	IF TimeElapsed > 0 THEN
		Speed_ips := (Distance/TimeElapsed);
		Speed_fps := Speed_ips/12;
		Speed_fpm := Speed_fps*60;
	END_IF
	IF TotalCounts > 0 THEN
		DistperCount := Distance / UDINT_TO_REAL(TotalCounts);
	END_IF
		Reading := FALSE;
END_IF

END_PROGRAM

// ---- FunctionBlocks/Binder/BinderX_ReleaseControl.TcPOU
PROGRAM BinderX_ReleaseControl
VAR
	BinderHoldFB: FB_Binder_SingulateHold;
	Binder_Pusher: FB_BinderPusher;

	Binder		:	ST_Binder;

	BinderDataIn AT %I*: ST_FromBinder;
	BinderDataOut AT %Q*: ST_ToBinder;
	BinderState AT %I*: ST_BinderState;
	
	// Dummy Points for Compiling
	dummyIn		:	BOOL;
	dummyOut	:	BOOL;
	OCRHoldFB: INT;
END_VAR

VAR_OUTPUT
	Online	AT %Q*	: BOOL; // Send Online state to Safety
END_VAR

VAR CONSTANT
	GRABBER1_OCCUPIED:	UINT  := 1;
	GRABBER2_OCCUPIED: 	UINT  := 2;
	HOLDER_OCCUPIED:		UINT  := 3;
	PINSTOP_OUT:			UINT  := 4;
	
	PAUSED:						UINT  := 0;
	PRODUCT_PRESENT:			UINT  := 1;
	PRODUCT_ENTERING_OCR:		UINT  := 2;
	PRODUCT_READY_TO_PROCESS:	UINT  := 3;
	OCR_FINISHED:				UINT  := 4;	
	PRODUCT_EXITING_OCR:		UINT  := 5;
	RETURN_CONVEYOR_CLEARING:	UINT  := 6;
	RETURN_CONVEYOR_BUSY:		UINT  := 7;
END_VAR

(*
	Commented lines indicate what type of data item should be used for the signaling
*)

BinderHoldFB(
	In_Pause:= NOT Binder.FromBinder.Online,
//	In_ConveyorRunning := Conveyors.P8030_VFD.IsRunning,
	In_ReturnConveyorClearTime:= T#250MS, 
//	In_Grabber_Auto := Solenoids.GR8030_1_Status.Sts_EquipmentState.StsAuto,
//	In_GrabberExtended := ProxSensors.PX_23661_Extended.Out,
//	In_GrabberRetracted := ProxSensors.PX_23641_Retracted.Out,
//	In_SV_GrabberExtend := GVL_IO.SOL_10_Extend,
//	In_SV_GrabberRetract := GVL_IO.SOL_10_Retract,
//	In_PinStop_1_Auto := Solenoids.PS8030_1_Status.Sts_EquipmentState.StsAuto,
//	In_PinStop_1_Extended := ProxSensors.PX_23701_Extended.Out,
//	In_PinStop_1_Retracted := ProxSensors.PX_23681_Retracted.Out,
//	In_SV_PinStop_1_Extend := GVL_IO.SOL_11_Extend,
//	In_SV_PinStop_1_Retract := GVL_IO.SOL_11_Retract,
//	In_Holder_Auto := Solenoids.PS8030_2_Status.Sts_EquipmentState.StsAuto,
//	In_HolderExtended := ProxSensors.PX_23501_Extended.Out,
//	In_HolderRetracted := ProxSensors.PX_23481_Retracted.Out,
//	In_SV_HolderExtend := GVL_IO.SOL_13_Extend,
//	In_SV_HolderRetract := GVL_IO.SOL_13_Retract,
//	In_PinStop_2_Auto := Solenoids.PS8030_2_Status.Sts_EquipmentState.StsAuto,
//	In_PinStop_2_Extended := ProxSensors.PX_23541_Extended.Out,
//	In_PinStop_2_Retracted := ProxSensors.PX_23521_Retracted.Out,
//	In_SV_PinStop_2_Extend := GVL_IO.SOL_12_Extend,
//	In_SV_PinStop_2_Retract := GVL_IO.SOL_12_Retract,
	IN_Binder_Finished:= BinderDataIn.ProcessingComplete, 
//	PE_Grabber:= PhotoEyes.PE_23241.Out_OnOffFltrd, 
//	PE_PinStop_1:= PhotoEyes.PE_23461.Out_OnOffFltrd, 
//	PE_Holder:= PhotoEyes.PE_23521.Out_OnOffFltrd, 
//	PE_BinderExit := PhotoEyes.PE_23621.Out_OffFltrd, 
//	PE_ReturnConveyorOccupied:= PhotoEyes.PE_23741.Out_OffFltrd, 
	Status=> BinderDataOut.StatusSingulator, 
	Status_Output=> );

// Update variable to OCR that product is held and ready to be processed
//BinderDataOut.ProductHeld := BinderHoldFB.Status.PRODUCT_READY_TO_PROCESS AND GVL_IO.SOL_13_Extend AND ProxSensors.PX_23501_Extended.OutOnFltrd;;

// Push product out  
//Binder_Pusher(PE_Pusher:= (GVL_IO.P8030_Status.Sts_IsRunning) AND (PhotoEyes.PE_23621.Out) AND BinderHoldFB.Status.PRODUCT_EXITING_OCR,
//	PushTime:= T#250MS, 
//	);

//Binder.State.VlvBankPower := GVL_IO.OCRVlvBankPwr;
//Binder.State.DumpValve := GVL_IO.BinderAirDump; 
//Binder.State.SystemEstopOK := GVL_IO.SystemEstopsOK;
Binder.FromBinder := BinderDataIn;
Binder.ToBinder := BinderDataOut;

Online := BinderDataIn.Online;

END_PROGRAM

// ---- FunctionBlocks/Binder/FB_Binder_SingulateHold.TcPOU
FUNCTION_BLOCK FB_Binder_SingulateHold
VAR_INPUT
	{attribute 'OPC.UA.DA' := '1'}
	In_ResetState				:	BOOL;		// Clear the current functional state of the Binder

	In_Pause					:	BOOL;
	In_ConveyorRunning			:	BOOL;
	In_ReturnConveyorClearTime	:	TIME;
	IN_Binder_Finished			:	BOOL;
	
	PE_Grabber					:	BOOL;
	PE_PinStop_1				:	BOOL;
	PE_Holder					:	BOOL;
	PE_BinderExit				:	BOOL;
	PE_ReturnConveyorOccupied	:	BOOL;  // Photo eye that detects product on rack return conveyor
	
	In_Grabber_Auto				:	BOOL;
	In_SV_GrabberExtend			:	BOOL;
	In_SV_GrabberRetract		:	BOOL;
	In_GrabberExtended			:	BOOL;
	In_GrabberRetracted			:	BOOL;

	In_PinStop_1_Auto			:	BOOL;
	In_SV_PinStop_1_Extend		:	BOOL;
	In_SV_PinStop_1_Retract		:	BOOL;
	In_PinStop_1_Extended		:	BOOL;
	In_PinStop_1_Retracted		:	BOOL;

	In_PinStop_2_Auto			:	BOOL;
	In_SV_PinStop_2_Extend		:	BOOL;
	In_SV_PinStop_2_Retract		:	BOOL;
	In_PinStop_2_Extended		:	BOOL;
	In_PinStop_2_Retracted		:	BOOL;

	In_Holder_Auto				:	BOOL;
	In_SV_HolderExtend			:	BOOL;
	In_SV_HolderRetract			:	BOOL;
	In_HolderExtended			:	BOOL;
	In_HolderRetracted			:	BOOL;
	
END_VAR
VAR_OUTPUT
	{attribute 'OPC.UA.DA' := '1'}
	Out_Homed					:	BOOL;
	{attribute 'OPC.UA.DA' := '1'}
	Out_Ready					:	BOOL;
	{attribute 'OPC.UA.DA' := '1'}
	Out_Running					:	BOOL;

	Out_Grabber_Ext				:	BOOL;
	Out_Grabber_Ret				:	BOOL;

	Out_PinStop_1_Ext			:	BOOL;
	Out_PinStop_1_Ret			:	BOOL;

	Out_PinStop_2_Ext			:	BOOL;
	Out_PinStop_2_Ret			:	BOOL;

	Out_Holder_Ext				:	BOOL;
	Out_Holder_Ret				:	BOOL;
	
	{attribute 'OPC.UA.DA' := '1'}
	Status						:	UINT;		// General Binder singulate and hold status
	Status_Output				:	UINT;		// Binder singulate pin stop and grabber status
	
END_VAR
VAR	
	StartUp						:	BOOL := TRUE;
	rReturnConveyorOccupied		:	R_TRIG;
	fReturnConveyorExit			:	F_TRIG;
	tofReleaseConveyorClearTimer:	TOF;
	rProductFinished			:	R_TRIG;
	fProductCleared				:	F_TRIG;
	
	rProductEntering			:	R_TRIG;
	fProductEntering			:	F_TRIG;
	rResetState					:	R_TRIG;
	
	tonHomeWait					:	TON := (PT := T#1S);
	tonReadyWait				:	TON := (PT := T#1S);
	tonRunningWait				:	TON := (PT := T#5S);

	// Extend and Retract controls
	Grabber_Extend				:	BOOL;
	Grabber_Retract				:	BOOL;
	PinStop_1_Extend			:	BOOL;
	PinStop_1_Retract			:	BOOL;
	Holder_Extend				:	BOOL;
	Holder_Retract				:	BOOL;
	PinStop_2_Extend			:	BOOL;
	PinStop_2_Retract			:	BOOL;
END_VAR

VAR CONSTANT
	// Output Status
	GRABBER_OCCUPIED			:	UINT  := 1;
	PINSTOP_1_OUT				:	UINT  := 2;
	HOLDER_OCCUPIED				:	UINT  := 3;
	PINSTOP_2_OUT				:	UINT  := 4;
	
	// Singulation Status
	PAUSED						:	UINT  := 0;
	PRODUCT_PRESENT				:	UINT  := 1;
	PRODUCT_ENTERING_BINDER		:	UINT  := 2;
	PRODUCT_READY_TO_PROCESS	:	UINT  := 3;
	BINDER_FINISHED				:	UINT  := 4;	
	PRODUCT_EXITING_BINDER		:	UINT  := 5;
	RETURN_CONVEYOR_CLEARING	:	UINT  := 6;
	RETURN_CONVEYOR_BUSY		:	UINT  := 7;
END_VAR

// Process the In_ResetState
rResetState(CLK:=In_ResetState);

IF rResetState.Q THEN
	// Clear the Status
	Status := 0;
	// Revert to the StartUp state
	StartUp := TRUE;
	// Revert to the NOT Homed state
	Out_Homed := FALSE;
	tonHomeWait(IN := FALSE);
	// Revert to the NOT Ready state
	Out_Ready := FALSE;
	tonReadyWait(IN := FALSE);
	// Revert to the NOT Running state
	Out_Running := FALSE;
	tonRunningWait(IN := FALSE);
	// Clear the reset request
	In_ResetState := FALSE;
END_IF

// Home the 
IF StartUp  OR NOT Out_Homed OR NOT Out_Ready THEN
	Status.PAUSED := TRUE;
	
	tonHomeWait.IN := NOT Out_Homed;
	tonHomeWait();
	IF NOT Out_Homed THEN
		// Grabber
		Grabber_Retract := TRUE;
		Grabber_Extend := FALSE;
		// PinStop_1
		PinStop_1_Retract := FALSE;
		PinStop_1_Extend := TRUE;
		// Holder
		Holder_Retract := TRUE;
		Holder_Extend := FALSE;
		// PinStop_2
		PinStop_2_Retract := FALSE;
		PinStop_2_Extend := TRUE;
		IF In_GrabberRetracted
		   AND In_PinStop_1_Extended
		   AND In_HolderRetracted
		   AND In_PinStop_2_Extended
		   THEN
			Out_Homed := tonHomeWait.Q;
		END_IF
	END_IF

	tonReadyWait.IN := NOT Out_Ready AND Out_Homed;
	tonReadyWait();
	IF NOT Out_Ready AND Out_Homed THEN
		// PinStop_1
		PinStop_1_Retract := FALSE;
		PinStop_1_Extend := TRUE;
		// PinStop_2
		PinStop_2_Retract := FALSE;
		PinStop_2_Extend := TRUE;
		IF In_GrabberRetracted
		   AND In_PinStop_1_Extended
		   AND In_HolderRetracted
		   AND In_PinStop_2_Extended
		   THEN
			Out_Ready := tonReadyWait.Q;
		END_IF
	END_IF

	StartUp := NOT Out_Homed OR NOT Out_Ready;
	Out_Running := FALSE;
	
ELSIF In_Pause OR NOT In_ConveyorRunning THEN
	// Grabber
	Grabber_Retract := FALSE;
	Grabber_Extend := FALSE;
	// PinStop_1
	PinStop_1_Retract := FALSE;
	PinStop_1_Extend := FALSE;
	// Holder
	Holder_Retract := FALSE;
	Holder_Extend := FALSE;
	// PinStop_2
	PinStop_2_Retract := FALSE;
	PinStop_2_Extend := FALSE;

ELSIF NOT Out_Running THEN
	tonRunningWait.IN := NOT OUT_Running AND Out_Ready AND Out_Homed AND In_ConveyorRunning;
	tonRunningWait();
	Out_Running := tonRunningWait.Q;
ELSIF Out_Running THEN
	Status.PAUSED := FALSE;

	a_EntryControl();
		
	a_ReleaseToBinder();
	
	a_HoldProduct();
	
	// Watch finished trigger to release product from
	rProductFinished(CLK:= IN_Binder_Finished);
	
	IF rProductFinished.Q THEN
		Status.BINDER_FINISHED := TRUE;
	END_IF
	
	// Watch release conveyor to make sure it is clear to release from OCR
	a_WatchReleaseConveyor();
		
	a_ReleaseFromBinder();
	
	fProductCleared(CLK:= PE_BinderExit AND Status.PRODUCT_EXITING_BINDER);
	
	// PinStop_2
	PinStop_2_Retract := Status.PRODUCT_EXITING_BINDER;
	PinStop_2_Extend := NOT Status.PRODUCT_EXITING_BINDER;
	IF fProductCleared.Q THEN
		Status.PRODUCT_EXITING_BINDER := FALSE;
//		IF Status.PRODUCT_PRESENT OR PE_PinStop_1 THEN
//			ReleaseToOCR();
//		END_IF
	END_IF
ELSE
	// Grabber
	Grabber_Retract := TRUE;
	Grabber_Extend := FALSE;
	// PinStop_1
	PinStop_1_Retract := FALSE;
	PinStop_1_Extend := TRUE;
	// Holder
	Holder_Retract := TRUE;
	Holder_Extend := FALSE;
	// PinStop_2
	PinStop_2_Retract := FALSE;
	PinStop_2_Extend := TRUE;
END_IF

// Activate all the outputs in one place
Status_Output.GRABBER_OCCUPIED := Grabber(Active := In_Grabber_Auto, Extend:= Grabber_Extend, Retract := Grabber_Retract);
Status_Output.HOLDER_OCCUPIED := Holder(Active := In_Holder_Auto, Extend:= Holder_Extend, Retract := Holder_Retract);
Status_Output.PINSTOP_1_OUT := PinStop_1(Active:= In_PinStop_1_Auto, Extend := PinStop_1_Extend, Retract:= PinStop_1_Retract);
Status_Output.PINSTOP_2_OUT := PinStop_2(Active:= In_PinStop_2_Auto, Extend := PinStop_2_Extend, Retract:= PinStop_2_Retract);

ACTION a_EntryControl:
(* Set PRODUCT_PRESENT when:
	PE_PinStop_1 is ON
	OR PRODUCT_ENTERRING_OCR is ON
*)
Status.PRODUCT_PRESENT := PE_PinStop_1 OR Status.PRODUCT_ENTERING_BINDER;
// Retract the Pin stop in response to the Release to the OCR, and the state of the Pin stop PE
rProductEntering(CLK:= Status.PRODUCT_ENTERING_BINDER);
IF rProductEntering.Q THEN
	PinStop_1_Extend := FALSE;
	PinStop_1_Retract := TRUE;
END_IF
fProductEntering(CLK := PE_PinStop_1);
IF fProductEntering.Q THEN
	PinStop_1_Extend := TRUE;
	PinStop_1_Retract := FALSE;
END_IF

// If the grabber recieves product while Product is physically or logically at Pin Stop 1, then hold it at the grabber

Grabber_Extend := (PE_Grabber AND Status.PRODUCT_PRESENT) OR Status.PRODUCT_ENTERING_BINDER;
Grabber_Retract := NOT Grabber_Extend;
END_ACTION

ACTION a_HoldProduct:
IF PE_Holder THEN
	Status.PRODUCT_PRESENT := FALSE;
	Status.PRODUCT_ENTERING_BINDER := FALSE;
	IF NOT Status.PRODUCT_EXITING_BINDER THEN
		Holder_Extend := TRUE;
		Holder_Retract := FALSE;
		Status.PRODUCT_READY_TO_PROCESS := TRUE;
	END_IF
END_IF
END_ACTION

ACTION a_ReleaseFromBinder:
IF Status.BINDER_FINISHED AND NOT(Status.RETURN_CONVEYOR_BUSY) THEN
	Status.PRODUCT_READY_TO_PROCESS := FALSE;
	Status.PRODUCT_EXITING_BINDER := TRUE;
	Status.BINDER_FINISHED := FALSE;
	// Holder
	Holder_Retract := TRUE;
	Holder_Extend := FALSE;
	// PinStop_2
	PinStop_2_Retract := TRUE;
	PinStop_2_Extend := FALSE;
END_IF
END_ACTION

ACTION a_ReleaseToBinder:
IF Status.PRODUCT_PRESENT 
   AND NOT(Status_Output.HOLDER_OCCUPIED)
   AND NOT(Status.PRODUCT_ENTERING_BINDER)
   AND NOT(Status.PRODUCT_EXITING_BINDER)  THEN
	Status.PRODUCT_ENTERING_BINDER := TRUE;
END_IF
END_ACTION

ACTION a_WatchReleaseConveyor:
rReturnConveyorOccupied(CLK:= PE_ReturnConveyorOccupied);

IF rReturnConveyorOccupied.Q THEN
	Status.RETURN_CONVEYOR_CLEARING := TRUE;
END_IF

fReturnConveyorExit(CLK:= Status.RETURN_CONVEYOR_BUSY AND PE_BinderExit);

IF fReturnConveyorExit.Q THEN
	Status.RETURN_CONVEYOR_CLEARING := FALSE;
END_IF

tofReleaseConveyorClearTimer(IN:= Status.RETURN_CONVEYOR_CLEARING, PT:= In_ReturnConveyorClearTime);

Status.RETURN_CONVEYOR_BUSY:= tofReleaseConveyorClearTimer.Q;
END_ACTION

METHOD Grabber : BOOL
VAR_INPUT
	Active	: BOOL;	
	Extend	: BOOL;
	Retract	: BOOL;
END_VAR
IF Active THEN
	IF Extend THEN
		Out_Grabber_Ext := TRUE;
		Out_Grabber_Ret := FALSE;
	ELSIF Retract THEN
		Out_Grabber_Ext := FALSE;
		Out_Grabber_Ret := TRUE;
	ELSE
		Out_Grabber_Ext := FALSE;
		Out_Grabber_Ret := FALSE;
	END_IF
ELSE
	Out_Grabber_Ext := FALSE;
	Out_Grabber_Ret := FALSE;
END_IF

Grabber := Out_Grabber_Ext OR In_GrabberExtended;
END_METHOD

METHOD Holder : BOOL
VAR_INPUT
	Active	: BOOL;
	Extend	: BOOL;
	Retract	: BOOL;
END_VAR
IF Active THEN
	IF Extend THEN
		Out_Holder_Ext := TRUE;
		Out_Holder_Ret := FALSE;
	ELSIF Retract THEN
		Out_Holder_Ext := FALSE;
		Out_Holder_Ret := TRUE;
	ELSE
		Out_Holder_Ext := FALSE;
		Out_Holder_Ret := FALSE;
	END_IF
ELSE
	Out_Holder_Ext := FALSE;
	Out_Holder_Ret := FALSE;
END_IF

Holder := Out_Holder_Ext OR In_HolderExtended;
END_METHOD

METHOD PinStop_1 : BOOL
VAR_INPUT
	Active	: BOOL;	
	Extend	: BOOL;
	Retract	: BOOL;
END_VAR
IF Active THEN
	IF Extend THEN
		Out_PinStop_1_Ext := TRUE;
		Out_PinStop_1_Ret := FALSE;
	ELSIF Retract THEN
		Out_PinStop_1_Ext := FALSE;
		Out_PinStop_1_Ret := TRUE;
	ELSE
		Out_PinStop_1_Ext := FALSE;
		Out_PinStop_1_Ret := FALSE;
	END_IF
ELSE
	Out_PinStop_1_Ext := FALSE;
	Out_PinStop_1_Ret := FALSE;
END_IF

PinStop_1 := Out_PinStop_1_Ext OR In_PinStop_1_Extended;
END_METHOD

METHOD PinStop_2 : BOOL
VAR_INPUT
	Active	: BOOL;
	Extend	: BOOL;
	Retract	: BOOL;
END_VAR
IF Active THEN
	IF Extend THEN
		Out_PinStop_2_Ext := TRUE;
		Out_PinStop_2_Ret := FALSE;
	ELSIF Retract THEN
		Out_PinStop_2_Ext := FALSE;
		Out_PinStop_2_Ret := TRUE;
	ELSE
		Out_PinStop_2_Ext := FALSE;
		Out_PinStop_2_Ret := FALSE;
	END_IF
ELSE
	Out_PinStop_2_Ext := FALSE;
	Out_PinStop_2_Ret := FALSE;
END_IF

PinStop_2 := Out_PinStop_2_Ext OR In_PinStop_2_Extended;
END_METHOD

END_FUNCTION_BLOCK

// ---- FunctionBlocks/Binder/FB_BinderPusher.TcPOU
FUNCTION_BLOCK FB_BinderPusher
VAR_INPUT
	PE_Pusher: BOOL;
	PushTime:	TIME;
END_VAR
VAR_OUTPUT
	Out_Pusher_Ext:	BOOL;
	Out_Pusher_Ret:	BOOL;
	PushingActive: BOOL;
END_VAR
VAR
	fPusher: F_TRIG;
	
	tonPusherArm: TON;
END_VAR

fPusher(CLK:= PE_Pusher);

IF fPusher.Q THEN
	Out_Pusher_Ext := TRUE;
	Out_Pusher_Ret := FALSE;
	PushingActive := TRUE;
END_IF

tonPusherArm(IN:=PushingActive , PT:= PushTime);

IF tonPusherArm.Q  THEN
	Out_Pusher_Ext := FALSE;
	Out_Pusher_Ret := TRUE;
	PushingActive := FALSE;
END_IF

END_FUNCTION_BLOCK

// ---- FunctionBlocks/FB_Merge/FB_Merge2.TcPOU
FUNCTION_BLOCK FB_Merge2
(* This function block can handle any number of Inlets to the merge by changing the constant "Cfg_MergeInletCount" 
	and then saving it as a new named function block. 
*)

VAR CONSTANT
	MERGEINLETCOUNT			:	INT := 2;		// Number of inlets on the merge
END_VAR

VAR_IN_OUT
	In_MergeProcessOrder	:	ARRAY [1..MERGEINLETCOUNT] OF INT;	// Processing order of the merge inlets
END_VAR

VAR_INPUT
	{attribute 'OPC.UA.DA' := '1'}
	In_MergeState				:	E_StateCntrl;	// The State of the merge take away conveyor
	In_MergeInletArry			:	ARRAY [1..MERGEINLETCOUNT] OF ST_MergeInlet;
	In_MergeTakeAwayMtrFdbk		:	BOOL;			// Merge Take Away Motor Feedback, 1=Running
	{attribute 'OPC.UA.DA' := '1'}
	In_PhotoEyeJamDetect		:	BOOL;			// Photo Eye located to detect jams at the assigned merge
	
	In_SimActive				:	BOOL;	
	In_Init						:	BOOL;
		
	In_MergeWakeTrigArry		: 	ARRAY [1..5] OF BOOL;
	Cfg_ClearTakeAwayTime		: 	REAL;
	{attribute 'OPC.UA.DA' := '1'}
	Cfg_MergeName				:	STRING(20);		// Name used to Identify the Merge on the HMI
	{attribute 'OPC.UA.DA' := '1'}
	Cfg_JammedTime				: 	REAL := 15;
END_VAR

VAR_OUTPUT
	Sts_MergeSts			:	ST_MergeSts;
	Sts_MergeInletStsArry	:	ARRAY [1..MERGEINLETCOUNT]OF ST_MergeInletSts;
END_VAR

VAR
	MergeRunOutActive		:	BOOL;
	MergeStateChanged		:	R_TRIG;	
	LastMergeState			: 	E_StateCntrl;

	MergeEnabledRTrig		: 	R_TRIG;
	MergeEnabledFTrig		: 	F_TRIG;
	inletindex				: 	INT := 0;
	processIndex			:	INT := 0;	
	i						:	INT;
	j						:	INT;
	fb_MergeEntryArry		:	ARRAY [1..MERGEINLETCOUNT]OF FB_MergeInlet;
	MergeGrantedOwner		:	INT := 0;	// The ID (index) of the inlet that has the merge granted control 
	MergeSubState_old		: 	INT;
	AnotherMergeReqIsWaiting: 	BOOL;
	HiHiMergeReqIsWaiting	: 	BOOL;
	HiHiIndex				: 	INT;
	MergeCntrl				: 	INT;

	ClearTakeawayDelay		: 	BOOL;
	ClearTakeAwayTimer		: 	TON;
	LastClearTakeAwayTime	: 	REAL;
	nClearTakeAwayTime		: 	UINT;
	tClearTakeAwayTime		: 	TIME;

	LastJammedTime			:	REAL;
	nJammedTime				:	UINT;
	tJammedTime				:	TIME;
	fb_JamDetect			:	FB_JamDetect;
	
	bIncIndex				:	BOOL;
END_VAR

// Initialize the Merge Here
IF In_Init THEN
	// Make sure the Processing Order doesn't have zeros in it
	FOR i := 1 TO MERGEINLETCOUNT DO
		IF In_MergeProcessOrder[i] = 0 THEN
			In_MergeProcessOrder[i] := i;
		END_IF
	END_FOR
	IF processIndex = 0 THEN
		processIndex := 1;
	END_IF
	Sts_MergeSts.MergeSubState := E_MergeState.stStopped;
	Sts_MergeSts.MergeSubStateTxt := 'Stopped';
	Sts_MergeSts.InletCount := MERGEINLETCOUNT;
	MergeGrantedOwner := In_MergeProcessOrder[1];
END_IF

// Calculate and set the timer values
// Clear take away timer
IF LastClearTakeAwayTime <> Cfg_ClearTakeAwayTime THEN
	LastClearTakeAwayTime := Cfg_ClearTakeAwayTime;
	nClearTakeAwayTime := REAL_TO_UINT(LastClearTakeAwayTime * 1000); 
	tClearTakeAwayTime := UINT_TO_TIME(nClearTakeAwayTime);
END_IF

// Product Jam Wait timer
IF LastJammedTime <> Cfg_JammedTime THEN
	LastJammedTime := Cfg_JammedTime;
	nJammedTime := REAL_TO_UINT(LastJammedTime * 1000); 
	tJammedTime := UINT_TO_TIME(nJammedTime);
END_IF

// Run the Jam Detection
fb_JamDetect(In_PE := In_PhotoEyeJamDetect
			, In_Status := Sts_MergeSts.MergeTakeAwayMtrActive
			, CFG_PEOKState := 0
			, JamDetTime := tJammedTime
			, JamDetected => Sts_MergeSts.MergeJammed);

// Set MergeEnabled to the Take Away conveyor Auto, or the take away running, for manual opertion
Sts_MergeSts.MergeEnabled := ((In_MergeState = E_StateCntrl.stAuto) OR In_MergeTakeAwayMtrFdbk);

// If merge is just enabled set operation
MergeEnabledRTrig(CLK:= Sts_MergeSts.MergeEnabled, Q=> );	

// Cause a Re-process of the state when the state changes
MergeStateChanged(CLK := (In_MergeState <> LastMergeState), Q=> );
// Capture the state change for the next pass 
LastMergeState := In_MergeState;

// Test for a Merge state change, or an enable trigger
IF MergeEnabledRTrig.Q OR MergeStateChanged.Q THEN
	CASE In_MergeState OF
		// Auto
		E_StateCntrl.stAuto:
			Sts_MergeSts.MergeSubState := E_MergeState.stClearTakeAway;
			Sts_MergeSts.MergeSubStateTxt := 'Clear Take Away';
		
		// Manual
		E_StateCntrl.stManual:
			Sts_MergeSts.MergeTakeAwayMtrActive := In_MergeTakeAwayMtrFdbk;
			inletindex := DINT_TO_INT(In_MergeProcessOrder[1]);
			Sts_MergeSts.MergeSubState := E_MergeState.stMergeManual;
			Sts_MergeSts.MergeSubStateTxt := 'Manual';
	END_CASE
END_IF

// If Merge enabled drops set states per condition
MergeEnabledFTrig(CLK:= Sts_MergeSts.MergeEnabled, Q=> );
IF  MergeEnabledFTrig.Q OR MergeStateChanged.Q THEN
	CASE In_MergeState OF
		// Offline
		E_StateCntrl.stOffline:
			Sts_MergeSts.MergeSubState := E_MergeState.stStopped;
			Sts_MergeSts.MergeSubStateTxt := 'Stopped';
		// Faulted
		E_StateCntrl.stFaulted:
			Sts_MergeSts.MergeSubState := E_MergeState.stStopped;
			Sts_MergeSts.MergeSubStateTxt := 'Faulted';
	END_CASE
END_IF

//  ===== Set Up Merge Control for merge sub parts =====

// Call inlet function blocks
FOR i := 1 TO MERGEINLETCOUNT DO
	fb_MergeEntryArry[i](In_MergeSubState:= Sts_MergeSts.MergeSubState, In_TakeAwayMtrSts:= Sts_MergeSts.MergeTakeAwayMtrActive, In_MergeInletInput:= In_MergeInletArry[i], Sts_MergeInlet=> Sts_MergeInletStsArry[i], In_MergeWakeTrig := In_MergeWakeTrigArry[i]);
END_FOR

// Turn OFF the increment Index boolean
bIncIndex := FALSE;

CASE Sts_MergeSts.MergeSubState OF	
	// Stopped
	E_MergeState.stStopped:
		Sts_MergeSts.MergeTakeAwayMtrActive := FALSE;
		
	// Clear Takeaway	
	E_MergeState.stClearTakeAway:
		ClearTakeawayDelay := TRUE;
		// Set Take Away Motor Output
		Sts_MergeSts.MergeTakeAwayMtrActive := ClearTakeawayDelay;
		
	
		IF ClearTakeAwayTimer.Q THEN
			ClearTakeawayDelay := FALSE;
			//MergeGrantedOwner := 0;
			MergeGrantedOwner := In_MergeProcessOrder[1];
			// Reset Inlets and merge
			FOR i := 1 TO MERGEINLETCOUNT DO
				fb_MergeEntryArry[i].In_MergeGranted := FALSE;
			END_FOR
			 fb_MergeEntryArry[1].In_MergeGranted := TRUE;
			IF processIndex = 0 THEN
				processIndex := 1;
			END_IF
			inletindex := In_MergeProcessOrder[processIndex];
			Sts_MergeSts.MergeSubState := E_MergeState.stMergeOperational;
			Sts_MergeSts.MergeSubStateTxt := 'Operational';
		END_IF
		
	// Operational
	E_MergeState.stMergeOperational:

		// Set the inletIndex to the inlet identified at the processIndex in the ProcessOrder
		inletindex := In_MergeProcessOrder[processIndex];

		// Set Take Away Motor Output
		Sts_MergeSts.MergeTakeAwayMtrActive := TRUE;
		
		// Clear the flags that may be set
		AnotherMergeReqIsWaiting := FALSE;
		HiHiMergeReqIsWaiting := FALSE;
		HiHiIndex := 0;
		MergeRunOutActive := FALSE;
		FOR j := 1 TO MERGEINLETCOUNT DO
			IF fb_MergeEntryArry[j].Sts_MergeInlet.MergeRequested AND MergeGrantedOwner <> j AND MergeGrantedOwner <> 0 THEN
				AnotherMergeReqIsWaiting := TRUE;
			END_IF
			IF fb_MergeEntryArry[j].Sts_MergeInlet.HiHiDetected THEN
				HiHiMergeReqIsWaiting := TRUE;
				HiHiIndex := j;
			END_IF
			IF fb_MergeEntryArry[j].Sts_MergeInlet.MergeRunOutActive THEN
				MergeRunOutActive := TRUE;
			END_IF
		END_FOR

		// Call individual merge inlets branches
		IF fb_MergeEntryArry[inletindex].Sts_MergeInlet.MergeRequested THEN
			// Prioritize the HiHi request
			IF HiHiMergeReqIsWaiting THEN
				IF inletindex <> HiHiIndex THEN
					inletindex := HiHiIndex;
				END_IF
			END_IF
			IF NOT MergeRunOutActive THEN
				IF (MergeGrantedOwner = 0) THEN
					MergeGrantedOwner := inletindex;
					fb_MergeEntryArry[inletindex].In_MergeGranted := TRUE;
				END_IF
			END_IF
		ELSE
			bIncIndex := TRUE;
		END_IF	
		IF MergeGrantedOwner <> 0 THEN	
			IF (AnotherMergeReqIsWaiting AND fb_MergeEntryArry[MergeGrantedOwner].Sts_MergeInlet.MergeComplete)
			   OR HiHiMergeReqIsWaiting
			   THEN
				// Reset Inlet and merge
				fb_MergeEntryArry[MergeGrantedOwner].In_MergeGranted := FALSE;
				MergeGrantedOwner := 0;
				bIncIndex := TRUE;
			END_IF
		END_IF
	// Manual mode	
	E_MergeState.stMergeManual:
		// Set the inletIndex to the inlet identified at the processIndex in the ProcessOrder
		inletindex := In_MergeProcessOrder[processIndex];

		// Set Take Away Motor Output
		Sts_MergeSts.MergeTakeAwayMtrActive := In_MergeTakeAwayMtrFdbk;
		
		// Call individual merge inlets branches
		IF fb_MergeEntryArry[inletindex].Sts_MergeInlet.MergeRequested THEN
			// Prioritize the HiHi request
			IF HiHiMergeReqIsWaiting THEN
				IF inletindex <> HiHiIndex THEN
					inletindex := HiHiIndex;
				END_IF
			END_IF
			IF NOT MergeRunOutActive THEN
				IF (MergeGrantedOwner = 0) THEN
					MergeGrantedOwner := inletindex;
					fb_MergeEntryArry[inletindex].In_MergeGranted := TRUE;
				END_IF
			END_IF
		ELSE
			bIncIndex := TRUE;
		END_IF		
		IF (AnotherMergeReqIsWaiting AND fb_MergeEntryArry[MergeGrantedOwner].Sts_MergeInlet.MergeComplete)
			   OR HiHiMergeReqIsWaiting
			   THEN
				// Reset Inlet and merge
				fb_MergeEntryArry[MergeGrantedOwner].In_MergeGranted := FALSE;
				MergeGrantedOwner := 0;
				bIncIndex := TRUE;
		END_IF
END_CASE

// Take Away Timer
ClearTakeAwayTimer(IN:= ClearTakeawayDelay, PT:= tClearTakeAwayTime, Q=> , ET=> );

// Increment the processIndex
IF bIncIndex THEN
	processIndex := processIndex + 1;
	bIncIndex := FALSE;
	// Reset index if necessary
	IF (processIndex > MERGEINLETCOUNT) THEN
		processIndex := 1;
	END_IF
END_IF

END_FUNCTION_BLOCK

// ---- FunctionBlocks/FB_Merge/Merge Inlet/FB_MergeInlet.TcPOU
FUNCTION_BLOCK FB_MergeInlet
VAR_INPUT
	In_MergeSubState		:	E_MergeState;
	In_TakeAwayMtrSts		:	BOOL;
	In_MergeInletInput		:	ST_MergeInlet;	
	In_MergeGranted			:	BOOL;		// Merge request has been accepted and allowed (1=merge allowed)
	In_MergeWakeTrig		:   BOOL;
END_VAR
VAR_OUTPUT
	Sts_MergeInlet			:	ST_MergeInletSts;
END_VAR
VAR
	MergeEntryHasProduct		: 	BOOL;
	MergeEntryHighTimer			: 	TON;		// Timer to watch High Photo Eye
	MergeEntryHiHiTimer			: 	TON;		// Timer to watch HiHi Photo Eye
	MergeRelPrdctWaitTimer		: 	TON;		// Timer to release product if waiting too long for full mark to be reached
	
	InletStateChanged			:	R_TRIG;	
	LastInletState				: 	E_StateCntrl;
	InletEnabled				:	BOOL;

	ProductReleaseCountFTrig	: 	F_Trig;
	ReleaseCountWaitTimer		: 	TON;
	ClearRunOutTimer			: 	TP;			// Run the timer for this long to clear out the merge
	fClearRunOut				:	F_TRIG;		// Detect when the ClearRunOut has completed
	ClearHiHiTimer				: 	TP;			// Run the timer for this long to clear a HiHi condition
	MergeRequestRTrig			: 	R_TRIG;
	RunEnable					: 	BOOL;
	MergePreLoad				: 	BOOL;
	MergeGrantedFTrig			: 	F_TRIG;
	ManualModeFTrig				: 	F_TRIG;
	ManualOperEnable			: 	BOOL;
	ManModeTrig					: 	R_TRIG;
	TimerReleaseCountWaitActive	:	BOOL;
	LastHighTriggerTime			:	REAL;
	LastHiHiTriggerTime			:	REAL;
	LastHiHiClearTime			:	REAL;
	LastMrgReqPrdctWaitTime		:	REAL;
	LastReleaseCountWaitTime	:	REAL;
	LastClearRunOutTime			:	REAL;

	nHighTriggerTime			:	UINT;
	nHiHiTriggerTime			:	UINT;
	nHiHiClearTime				:	UINT;
	nMrgReqPrdctWaitTime		:	UINT;
	nReleaseCountWaitTime		:	UINT;
	nClearRunOutTime			:	UINT;

	tHighTriggerTime			:	TIME;
	tHiHiTriggerTime			:	TIME;
	tHiHiClearTime				:	TIME;
	tMrgReqPrdctWaitTime		:	TIME;
	tReleaseCountWaitTime		:	TIME;
	tClearRunOutTime			:	TIME;
END_VAR

// Calculate and set the timer values
// High Water Mark trigger timer
IF LastHighTriggerTime <> In_MergeInletInput.Cfg.Cfg_HighTriggerTime THEN
	LastHighTriggerTime := In_MergeInletInput.Cfg.Cfg_HighTriggerTime;
	nHighTriggerTime := REAL_TO_UINT(LastHighTriggerTime * 1000); 
	tHighTriggerTime := UINT_TO_TIME(nHighTriggerTime);
END_IF

// HiHi Water Mark trigger timer
IF LastHiHiTriggerTime <> In_MergeInletInput.Cfg.Cfg_HiHiTriggerTime THEN
	LastHiHiTriggerTime := In_MergeInletInput.Cfg.Cfg_HiHiTriggerTime;
	nHiHiTriggerTime := REAL_TO_UINT(LastHiHiTriggerTime * 1000); 
	tHiHiTriggerTime := UINT_TO_TIME(nHiHiTriggerTime);
END_IF

// HiHi Water Mark clear timer
IF LastHiHiClearTime <> In_MergeInletInput.Cfg.Cfg_HiHiClearTime THEN
	LastHiHiClearTime := In_MergeInletInput.Cfg.Cfg_HiHiClearTime;
	nHiHiClearTime := REAL_TO_UINT(LastHiHiClearTime * 1000); 
	tHiHiClearTime := UINT_TO_TIME(nHiHiClearTime);
END_IF

// Product Wait timer
IF LastMrgReqPrdctWaitTime <> In_MergeInletInput.Cfg.Cfg_MrgReqPrdctWaitTime THEN
	LastMrgReqPrdctWaitTime := In_MergeInletInput.Cfg.Cfg_MrgReqPrdctWaitTime;
	nMrgReqPrdctWaitTime := REAL_TO_UINT(LastMrgReqPrdctWaitTime * 1000); 
	tMrgReqPrdctWaitTime := UINT_TO_TIME(nMrgReqPrdctWaitTime);
END_IF

// Fulfilled Release Count Wait timer
IF LastReleaseCountWaitTime <> In_MergeInletInput.Cfg.Cfg_ReleaseCountWaitTime THEN
	LastReleaseCountWaitTime := In_MergeInletInput.Cfg.Cfg_ReleaseCountWaitTime;
	nReleaseCountWaitTime := REAL_TO_UINT(LastReleaseCountWaitTime * 1000); 
	tReleaseCountWaitTime := UINT_TO_TIME(nReleaseCountWaitTime);
END_IF

// Run-Out Clear timer
IF LastClearRunOutTime <> In_MergeInletInput.Cfg.Cfg_ClearRunOutTime THEN
	LastClearRunOutTime := In_MergeInletInput.Cfg.Cfg_ClearRunOutTime;
	nClearRunOutTime := REAL_TO_UINT(LastClearRunOutTime * 1000); 
	tClearRunOutTime := UINT_TO_TIME(nClearRunOutTime);
END_IF

// Set InletEnabled to the Inlet conveyor Auto, or the Inlet conveyor running (for manual opertion)
InletEnabled := ((In_MergeInletInput.Ctrl.In_InletState = E_StateCntrl.stAuto)
				OR (In_MergeInletInput.Ctrl.In_InletState = E_StateCntrl.stManual AND In_MergeInletInput.Ctrl.In_oMergeRelease));

// Watch for manual mode and manual PB
IF In_MergeSubState = E_MergeState.stMergeManual AND InletEnabled THEN
	ManualOperEnable := In_MergeInletInput.Ctrl.In_oMergeRelease;
ELSE
	ManualOperEnable := FALSE;
END_IF

ManualModeFTrig(CLK:= ManualOperEnable, Q=> );

// Look at photo eyes and determine if a merge request is needed
MergeEntryHasProduct:= (In_MergeSubState = E_MergeState.stMergeOperational)
 						AND In_MergeInletInput.Ctrl.PhotoEyeDischarge
						AND (In_MergeInletInput.Ctrl.In_InletState = E_StateCntrl.stAuto);
// Set timer to keep product from waiting too long if full mark is not met
MergeRelPrdctWaitTimer(IN:= MergeEntryHasProduct AND (In_MergeInletInput.Cfg.Cfg_UseHighWaterPE OR In_MergeInletInput.Cfg.Cfg_UseHiHiWaterPE)
						, PT:= tMrgReqPrdctWaitTime, Q=> , ET=> );

// Watch the Timer to check for a High Water event
MergeEntryHighTimer.IN:= In_MergeInletInput.Ctrl.PhotoEyeEntryHigh AND In_MergeInletInput.Cfg.Cfg_UseHighWaterPE AND MergeEntryHasProduct;
MergeEntryHighTimer(PT:= tHighTriggerTime, Q=> , ET=> );

// Watch the Timer to check for a HiHi Water event
MergeEntryHighTimer.IN:= In_MergeInletInput.Ctrl.PhotoEyeEntryHiHi AND In_MergeInletInput.Cfg.Cfg_UseHiHiWaterPE AND MergeEntryHasProduct;
MergeEntryHiHiTimer(PT:= tHiHiTriggerTime, Q=> , ET=> );
IF (MergeEntryHiHiTimer.Q) THEN
	Sts_MergeInlet.HiHiDetected := MergeEntryHiHiTimer.Q;
END_IF

// Set merge request based on entry and full PE's and wait timer(s)
IF ((MergeEntryHighTimer.Q)
   OR (MergeEntryHiHiTimer.Q)
   OR ((NOT In_MergeInletInput.Cfg.Cfg_UseHighWaterPE AND NOT In_MergeInletInput.Cfg.Cfg_UseHiHiWaterPE) AND MergeEntryHasProduct)
   OR (MergeRelPrdctWaitTimer.Q)) 
   AND (NOT Sts_MergeInlet.MergeRequested AND NOT In_MergeGranted) OR ManualOperEnable THEN
	Sts_MergeInlet.MergeRequested := TRUE;
ELSIF Sts_MergeInlet.MergeRequested AND (NOT MergeEntryHasProduct) AND (NOT In_MergeGranted) THEN
	Sts_MergeInlet.MergeRequested := FALSE;
ELSIF In_MergeGranted THEN
	Sts_MergeInlet.MergeRequested := FALSE;
END_IF

// Upon merge request or entry of manual mode reset Count, Timer and Complete bit
ManModeTrig(CLK:= In_MergeSubState = E_MergeState.stMergeManual, Q=> );
MergeRequestRTrig(CLK:= Sts_MergeInlet.MergeRequested, Q=> );
IF MergeRequestRTrig.Q OR ManModeTrig.Q THEN
	Sts_MergeInlet.CrrntReleaseCount := 0;
	Sts_MergeInlet.MergeComplete := FALSE;
//	ManualOperEnable := FALSE;
END_IF

// If merge granted and HiHi Water mark detected, run the merge for the HiHi Clear time
//	This is a Timer Pulse so it will run for a specified period of time after the rising edge of the In condition is detected 
ClearHiHiTimer(IN := Sts_MergeInlet.HiHiDetected AND In_MergeGranted, PT := tHiHiClearTime);
	
// If merge granted count product release on falling trigger of the photo eye
//	Don't add up the count if the ClearRunOutTimer is running
ProductReleaseCountFTrig(CLK:= In_MergeInletInput.Ctrl.PhotoEyeDischarge, Q=> );
IF ProductReleaseCountFTrig.Q AND In_MergeGranted AND NOT ClearRunOutTimer.Q THEN
	Sts_MergeInlet.CrrntReleaseCount := Sts_MergeInlet.CrrntReleaseCount +1; 
END_IF

// If merge granted set timer to release if count isn't met
// Restart/stop the count when the merge is complete, a manual release is in process, an item is detected at the merge discharge
TimerReleaseCountWaitActive := In_MergeGranted AND Sts_MergeInlet.Sts_MergeInletRun 
											AND (NOT Sts_MergeInlet.MergeComplete) 
											AND (NOT ManualOperEnable) 
											AND (NOT MergeEntryHasProduct);
ReleaseCountWaitTimer(IN:= TimerReleaseCountWaitActive, PT:= tReleaseCountWaitTime, Q=> , ET=> );

// Set to complete if release count is met or if count wait timer expires 
IF ((In_MergeGranted AND In_TakeAwayMtrSts)
   AND NOT ManualOperEnable 
   AND NOT ClearHiHiTimer.Q 
   AND ((Sts_MergeInlet.CrrntReleaseCount >= In_MergeInletInput.Cfg.Cfg_ReleaseCount 
   		AND In_MergeInletInput.Cfg.Cfg_ReleaseCount >= 0) 
   		OR ReleaseCountWaitTimer.Q))
   OR ManualModeFTrig.Q 
   THEN
	Sts_MergeInlet.MergeComplete := TRUE;
END_IF

// Set the HiHiTimedReleaseActive when the merge is granted and the a HiHi Event was detected
Sts_MergeInlet.HiHiTimedReleaseActive := ClearHiHiTimer.Q;

// Reset Complete when merge granted is released
// Clear the Release count
// Set the RunOutActive flag to prevent jams while the last released item is cleared into the merge
MergeGrantedFTrig(CLK:= In_MergeGranted, Q=> );
IF MergeGrantedFTrig.Q THEN
	Sts_MergeInlet.MergeRunOutActive := TRUE;
	Sts_MergeInlet.CrrntReleaseCount := 0;
	Sts_MergeInlet.MergeComplete := FALSE;
	Sts_MergeInlet.HiHiDetected := FALSE;
END_IF

// Start the ClearRunOutTimer when the MergeRunOutActive is on and the Discharge PE is clear
ClearRunOutTimer(IN:= Sts_MergeInlet.MergeRunOutActive AND NOT In_MergeInletInput.Ctrl.PhotoEyeDischarge, PT := tClearRunOutTime);

// Use the ClearRunOutTimer to reset the MergeRunOutActive
fClearRunOut(CLK := ClearRunOutTimer.Q);
IF fClearRunOut.Q THEN
	Sts_MergeInlet.MergeRunOutActive := FALSE;
END_IF
 
MergePreLoad := (NOT In_MergeGranted) AND (NOT In_MergeInletInput.Ctrl.PhotoEyeDischarge);	

// Set Run Output, whatever it involves
RunEnable := In_MergeSubState = E_MergeState.stMergeOperational AND In_TakeAwayMtrSts AND (In_MergeGranted
		OR MergePreLoad) OR (ManualOperEnable AND In_MergeGranted);
Sts_MergeInlet.Out_MergeInletRunActive := RunEnable AND (NOT In_MergeInletInput.Ctrl.SimActive);
 
Sts_MergeInlet.Sts_MergeInletRun := (In_MergeInletInput.Cfg.Cfg_UseMtrFdBck AND In_MergeInletInput.Ctrl.MergeInletMtrFdBck) OR ((NOT In_MergeInletInput.Cfg.Cfg_UseMtrFdBck) AND RunEnable);

// Indicate the Granted condition
Sts_MergeInlet.Granted := In_MergeGranted;

END_FUNCTION_BLOCK

// ---- FunctionBlocks/FB_Merge/MergeExample.TcPOU
PROGRAM MergeExample
VAR CONSTANT
	// Change this to Match the number of inlets to ther merge, and create one constant per merge
	MERGEINLETCOUNT				:	DINT := 2;
END_VAR

VAR PERSISTENT
	// This array is used by the HMI to configure each merge inlet
	//	The items in this array can also be configured in the execution portion of the code, as shown in this example
	MergeTestInletCfgArray		:	ARRAY[1..MERGEINLETCOUNT] OF ST_MergeInletCfg;
	// This array allows the processing order of the inlets to be customized
	MergeTestProcessingOrder	:	ARRAY[1..MERGEINLETCOUNT] OF INT;
END_VAR

VAR
	// The ignition faceplate expexts the data items associated with this merge to all begin with the name assigned to the FB_MergeX instance
	MergeTest					:	FB_Merge2;
	MergeTestInletArray			:	ARRAY[1..MERGEINLETCOUNT] OF ST_MergeInlet;
	MergeTestInletStsArry		:	ARRAY[1..MERGEINLETCOUNT] OF ST_MergeInletSts;
	MergeTestWakeTrigArry		:	ARRAY[1..5] OF BOOL;
	MergeTestSts				:	ST_MergeSts;

	// These data items exist for testing purposes only
	MergeTestState				:	E_StateCntrl;
	MergeTestTakeAwayMtrFdbk	:	BOOL;
	SimActive					:	BOOL;
END_VAR

// Set-up the Merge Inlets
// Merge Inlet 1 Configuration
//	These items can also be configured in the Ignition Faceplate
//	The time items are REAL data types and are multipled by 1000 so they can have a resolution of 1 ms if desired
//	The MergeName is a 20 character string
//	The Use items are booleans and the ON state indicates they will be processed
MergeTestInletCfgArray[1].Cfg_ClearRunOutTime := 10;
MergeTestInletCfgArray[1].Cfg_HighTriggerTime := 1;
MergeTestInletCfgArray[1].Cfg_HiHiClearTime := 20;
MergeTestInletCfgArray[1].Cfg_HiHiTriggerTime := 5;
MergeTestInletCfgArray[1].Cfg_MrgReqPrdctWaitTime := 5;
MergeTestInletCfgArray[1].Cfg_ReleaseCount := 10;
MergeTestInletCfgArray[1].Cfg_ReleaseCountWaitTime := 2;
MergeTestInletCfgArray[1].Cfg_MergeName := 'Dock Door 1';
MergeTestInletCfgArray[1].Cfg_UseHighWaterPE := FALSE;
MergeTestInletCfgArray[1].Cfg_UseHiHiWaterPE := FALSE;
MergeTestInletCfgArray[1].Cfg_UseMtrFdBck := FALSE;

// This statement assigns the Persistent Data items to the MergeInletArray configuration item
//	It allows the configuration items to be persistent, without making the whole array be persistent
MergeTestInletArray[1].Cfg := MergeTestInletCfgArray[1];
// Controls the simulation state of the merge inlet
MergeTestInletArray[1].Ctrl.SimActive := SimActive;

// Merge Inlet 2
MergeTestInletCfgArray[2].Cfg_ClearRunOutTime := 10;
MergeTestInletCfgArray[2].Cfg_HighTriggerTime := 1;
MergeTestInletCfgArray[2].Cfg_HiHiClearTime := 20;
MergeTestInletCfgArray[2].Cfg_HiHiTriggerTime := 5;
MergeTestInletCfgArray[2].Cfg_MergeName := 'Dock Door 2';
MergeTestInletCfgArray[2].Cfg_MrgReqPrdctWaitTime := 5;
MergeTestInletCfgArray[2].Cfg_ReleaseCount := 10;
MergeTestInletCfgArray[2].Cfg_ReleaseCountWaitTime := 2;
MergeTestInletCfgArray[2].Cfg_UseHighWaterPE := FALSE;
MergeTestInletCfgArray[2].Cfg_UseHiHiWaterPE := FALSE;
MergeTestInletCfgArray[2].Cfg_UseMtrFdBck := FALSE;

MergeTestInletArray[2].Cfg := MergeTestInletCfgArray[2];
MergeTestInletArray[2].Ctrl.SimActive := SimActive;

// Execute the Merge Logic
MergeTest(In_MergeState := MergeTestState
			, In_MergeInletArry := MergeTestInletArray
			, In_MergeProcessOrder := MergeTestProcessingOrder
			, In_MergeTakeAwayMtrFdbk := MergeTestTakeAwayMtrFdbk
			, In_SimActive := SimActive
			, In_Init := GVL_IO.INIT
			, In_MergeWakeTrigArry := MergeTestWakeTrigArry
			, Cfg_ClearTakeAwayTime := 10
			, Cfg_MergeName := 'Test'
			, Sts_MergeSts => MergeTestSts
			, Sts_MergeInletStsArry => MergeTestInletStsArry);

END_PROGRAM

// ---- FunctionBlocks/FB_MotionMerge/FB_MotionMerge.TcPOU
FUNCTION_BLOCK FB_MotionMerge
VAR_IN_OUT
	InOut_ConveyorArry: ARRAY[*] OF ST_MotionMergeItem; // Array for the total items on conveyor
END_VAR
VAR_INPUT
	{attribute 'OPC.UA.DA' := '1'}
	In_InductPhotoEye: BOOL;
	{attribute 'OPC.UA.DA' := '1'}
	In_DownstreamClearPhotoEye: BOOL;
	In_St_Encoder: ST_Encoder;
	{attribute 'OPC.UA.DA' := '1'}
	In_MergeRunning: BOOL;

	cfg_MotionMerge:	ST_MotionMergeConfig;
END_VAR

VAR_OUTPUT
	{attribute 'OPC.UA.DA' := '1'}
	Out_MergeSpaceBusy: BOOL;
	{attribute 'OPC.UA.DA' := '1'}
	Out_MergeClearing: BOOL;
END_VAR

VAR
	MergeStartedTrig: R_TRIG;
	LastMergeClearTime:	REAL;
	nMergeClearTime: UINT;
	Cfg_MergeClearTime: TIME := T#10S;
	ClearMergeTimer: TOF;
	ClearingMergeTakeAwayTimer: TON;
	InductPE_Rtrig: R_TRIG;
	InductPE_Ftrig: F_TRIG;
	ConveyorIndx: INT := 1;		// Index to add item to conveyor
	EncoderRead_Old: UDINT;
	i: INT;		// Index to process items on conveyor
	NextI: INT;		// Index of next to process items on conveyor
	GapSize: UDINT;
	InMergeSpace: BOOL;
	Distance_ItemStart: UDINT;
	Distance_ItemEnd: UDINT;
	Distance_ClearItemArry: UDINT;
	ArrayMinSize : DINT;
	ArrayMaxSize : DINT;
	EncoderMax	: UDINT;
END_VAR

// Set triggers for the rise and fall of the photoeye
InductPE_Rtrig(CLK:= In_InductPhotoEye, Q=> );
InductPE_Ftrig(CLK:= In_InductPhotoEye, Q=> );

// Calculate and set the merge clear timer
IF LastMergeClearTime <> cfg_MotionMerge.MergeClearTime THEN
	LastMergeClearTime := cfg_MotionMerge.MergeClearTime;
	nMergeClearTime := REAL_TO_UINT(LastMergeClearTime * 1000); 
	Cfg_MergeClearTime := UINT_TO_TIME(nMergeClearTime);
END_IF

IF EncoderMax = 0 THEN
	EncoderMax := LREAL_TO_UDINT(EXPT(2,In_ST_Encoder.BitMaskSize));
END_IF
// If rising take read of location on conveyor
IF InductPE_Rtrig.Q THEN
	InOut_ConveyorArry[ConveyorIndx].Count_InductStart := In_St_Encoder.CurrentCount;
//	InOut_ConveyorArry[ConveyorIndx].Count_InductStart := F_CalculateIndex(Offset := - UINT_TO_LINT(Cfg_MotionMerge.Item_ExtendFwd)
//																			, InitialValue := In_St_Encoder.CurrentCount
//																			, BufferSize := EncoderMax);
END_IF
ArrayMinSize := LOWER_BOUND(InOut_ConveyorArry,1);
ArrayMaxSize := UPPER_BOUND(InOut_ConveyorArry,1);
// If falling take read of location on conveyor and calculate length, comparing the magnitude of the start and end to get the absolute difference
IF InductPE_Ftrig.Q THEN
	InOut_ConveyorArry[ConveyorIndx].Count_InductEnd := In_St_Encoder.CurrentCount;
//	InOut_ConveyorArry[ConveyorIndx].Count_InductEnd := F_CalculateIndex(Offset := UINT_TO_LINT(Cfg_MotionMerge.Item_ExtendRev)
//																			, InitialValue := In_St_Encoder.CurrentCount
//																			, BufferSize := EncoderMax);
	InOut_ConveyorArry[ConveyorIndx].Length := F_CalculateDifference(CurrentIndex := InOut_ConveyorArry[ConveyorIndx].Count_InductEnd,
																	CompareIndex := InOut_ConveyorArry[ConveyorIndx].Count_InductStart,
																	BufferSize := EncoderMax);
	InOut_ConveyorArry[ConveyorIndx].OnConveyor := TRUE;
	ConveyorIndx := F_IncIndex(IDX:= ConveyorIndx , IdxMIN:= DINT_TO_INT(ArrayMinSize), IdxMAX:=DINT_TO_INT(ArrayMaxSize));
END_IF

// If conveyor has moved watch location of each item on conveyor and process accordingly
IF EncoderRead_Old <> In_St_Encoder.CurrentCount THEN
	FOR i := DINT_TO_INT(ArrayMinSize) TO DINT_TO_INT(ArrayMaxSize) DO	// array of items on conveyor with a limit of ARRAYSIZE_MAX
		IF InOut_ConveyorArry[i].OnConveyor = TRUE THEN // Only process if it is currently on the conveyor
			// Calculate distance of Item to merge point
			
//			Distance_ItemStart := InOut_ConveyorArry[i].Count_InductStart + Cfg_MotionMerge.MergeDistance - Cfg_MotionMerge.Item_ExtendFwd;
			Distance_ItemStart := F_CalculateIndex(Offset :=  (Cfg_MotionMerge.MergeDistance - Cfg_MotionMerge.Item_ExtendFwd)
													, InitialValue := InOut_ConveyorArry[i].Count_InductStart
													, BufferSize := EncoderMax);
//			Distance_ItemEnd := InOut_ConveyorArry[i].Count_InductEnd + Cfg_MotionMerge.MergeDistance + Cfg_MotionMerge.Item_ExtendRev;
			Distance_ItemEnd := F_CalculateIndex(Offset :=  (Cfg_MotionMerge.MergeDistance + Cfg_MotionMerge.Item_ExtendRev)
													, InitialValue := InOut_ConveyorArry[i].Count_InductEnd
													, BufferSize := EncoderMax);

			// If item is at merge point report that it is busy
			// Test for both possible start/end value conditions
			//	Start < End and Start > End
			IF (Distance_ItemEnd > Distance_ItemStart) THEN
				IF (In_St_Encoder.CurrentCount >= Distance_ItemStart) AND (In_St_Encoder.CurrentCount < Distance_ItemEnd)  THEN
					Out_MergeSpaceBusy := TRUE;
				END_IF
			ELSE
				IF (In_St_Encoder.CurrentCount >= Distance_ItemStart) OR (In_St_Encoder.CurrentCount < Distance_ItemEnd)  THEN
					Out_MergeSpaceBusy := TRUE;
				END_IF
			END_IF
			
			// If Item is past the merge or there is nothing behind it then report clear, otherwise look at opening to see if item will fit			
			// Test for when the Item End is greater than the Item start and when the Item Start is greater than the Item End
			//		If the CurrentCount is less than the ItemStart when the Currentcount is greater than the Item End, the Start is greater than the end
			IF (In_St_Encoder.CurrentCount > Distance_ItemEnd)
			   AND ((Distance_ItemEnd > Distance_ItemStart) OR (In_St_Encoder.CurrentCount < Distance_ItemStart))
			   THEN
				Nexti := F_IncIndex(IDX:= i , IdxMIN:= DINT_TO_INT(ArrayMinSize), IdxMAX:=DINT_TO_INT(ArrayMaxSize));
				IF (InOut_ConveyorArry[Nexti].OnConveyor = FALSE) THEN
					Out_MergeSpaceBusy := FALSE;
				ELSE
//					GapSize := InOut_ConveyorArry[Nexti].Count_InductStart - InOut_ConveyorArry[i].Count_InductEnd;	
					GapSize := F_CalculateDifference(CurrentIndex := (UDINT_TO_DINT(InOut_ConveyorArry[Nexti].Count_InductStart))
													, CompareIndex := InOut_ConveyorArry[i].Count_InductEnd
													, BufferSize := EncoderMax);	
				END_IF
					
				IF (GapSize > Cfg_MotionMerge.MergeOpening_Min) THEN  // If we had an encoder on the spur or the size of the item on the spur we could compare here ie: AND (GapSize > ItemToMerge)  
					Out_MergeSpaceBusy := FALSE;	
				END_IF		
			END_IF
		END_IF
		
		// Clear out items from the conveyor array
		Distance_ClearItemArry := F_CalculateDifference(CurrentIndex := In_St_Encoder.CurrentCount
													, CompareIndex := InOut_ConveyorArry[i].Count_InductStart
													, BufferSize := EncoderMax);
		IF (Distance_ClearItemArry > cfg_MotionMerge.MergeClearDistance) THEN
			InOut_ConveyorArry[i].OnConveyor := FALSE;
			InOut_ConveyorArry[i].Count_InductStart :=0;
			InOut_ConveyorArry[i].Count_InductEnd :=0;
			InOut_ConveyorArry[i].Length :=0;
		END_IF
		
	END_FOR
	
	EncoderRead_Old := In_St_Encoder.CurrentCount;
END_IF

	(* ------------------------------------------------------------------------------------
	Set up a clear timer interlock and watch to see if downstream is full and hold back merge items
	*)
	MergeStartedTrig(CLK:= In_MergeRunning);
	IF MergeStartedTrig.Q OR In_DownstreamClearPhotoEye THEN
		Out_MergeClearing := TRUE;
	END_IF
	
	ClearingMergeTakeAwayTimer(IN:= (Out_MergeClearing AND NOT In_DownstreamClearPhotoEye) , PT:= Cfg_MergeClearTime);
	IF ClearingMergeTakeAwayTimer.Q THEN
		Out_MergeClearing := FALSE;
	END_IF
	(*------------------------------------------------------------------------------------*)

END_FUNCTION_BLOCK

// ---- FunctionBlocks/Utils/F_CalculateDifference.TcPOU
(*
	This function calculates the difference between two indices using the max array size.
	This allows you to easily treat the array like a ring buffer
	For this function to work properly, the following rules MUST be observed
	1) CurrentIndex, CompareIndex and BufferSize are all unsigned
	3) BufferSize is the number of elements in an array, not the maximum array index
		An array defined as ARRAY[0..10] has 11 elements, not 10, as the maximum element implies
		If the array is defined as [0..ARRAYMAX], where ARRAYMAX is a constant, BufferSize = ARRAYMAX + 1
*)
FUNCTION F_CalculateDifference : UDINT 
VAR_INPUT
	CurrentIndex	: UDINT; //The offset that you want to calculate, the sign in important to indicate direction
	CompareIndex	: UDINT; //The original point in the array you want to evaluate
	BufferSize		: UDINT; //The size of the array, not the index of the last array element
END_VAR
VAR
	TempDifference	: UDINT;
END_VAR

(*
	Test the Compare and Current index values. If the CurrentIndex value is less than the CompareIndex,
	 assume that the Unsigned count has rolled to zero and adjust the distance accordingly
*)
// Test the TempIndex to determine what the return index should be
// If it is zero or greater, test against the BufferSize value
IF CurrentIndex < CompareIndex THEN
	TempDifference := BufferSize - CompareIndex;
	F_CalculateDifference := TempDifference + CurrentIndex;
ELSE
	// Return the Difference
	f_CalculateDifference := CurrentIndex - CompareIndex;
END_IF

END_FUNCTION

// ---- FunctionBlocks/Utils/F_IncIndex.TcPOU
FUNCTION F_IncIndex : INT
VAR_INPUT
	IDX:	INT;		// Index to be incremented
	IdxMIN:	INT;		// Min Value for index	
	IdxMAX:	INT;		// Max Value for index
END_VAR
VAR
END_VAR

IF IDX < IdxMAX THEN
	F_IncIndex := IDX + 1; 
ELSIF IDX = IdxMAX THEN
	F_IncIndex := IdxMIN;
ELSIF IDX < IdxMIN OR IDX > IdxMAX THEN
	F_IncIndex := IdxMIN;
END_IF

END_FUNCTION

// ---- FunctionBlocks/FB_MotionMerge/MotionMergeExample.TcPOU
PROGRAM MotionMergeExample
VAR
	bSimulate					: BOOL := FALSE;	// Indicates when runing a simulation
	Merge_1				: FB_MotionMerge;
	Merge_1MergeItemArry: ARRAY[MERGEARRAYSIZE_MIN..MERGEARRAYSIZE_MAX] OF ST_MotionMergeItem; // Array for the total items on conveyor
	st_MergeEncoder		: ST_Encoder;
	fb_MergeEncoder		: FB_ProcessEncoder;
	ENC_Raw				:	UINT;
END_VAR

VAR PERSISTENT
	Merge_1_Config				: ST_MotionMergeConfig; 
END_VAR

VAR CONSTANT
	MERGEMASKSIZE		: UINT := 16;	// Number of bits to mask into the Encoder Count, will define the size of the SORTERENCODERMAX value
	MERGEARRAYSIZE_MAX	: INT := 50;  // Number of items that are proccesed on conveyor at one time
	MERGEARRAYSIZE_MIN	: INT := 1;
END_VAR

// Setup and process the Merge Encoder
st_MergeEncoder.EncoderRawCount := ENC_Raw;
st_MergeEncoder.BitMaskSize := MERGEMASKSIZE;
fb_MergeEncoder(Encoder := st_MergeEncoder, Simulate :=bSimulate);

// Run Merge Logic
Merge_1(
	InOut_ConveyorArry := Merge_1MergeItemArry,
//	In_InductPhotoEye := Photoeyes.PE_22141.Out_OffFltrd,
	In_St_Encoder := st_MergeEncoder,
//	In_MergeRunning := Conveyors.P8005_VFD.IsRunning,
//	In_DownstreamClearPhotoEye := Photoeyes.PE_22081.JamDetected,
	cfg_MotionMerge := Merge_1_Config);

END_PROGRAM

// ---- FunctionBlocks/LEDControl/FB_LEDModeCtrl.TcPOU
FUNCTION_BLOCK FB_LEDModeCtrl
VAR_INPUT
	In_Light_Mode:	BYTE;		// Mode the light is in (0=Off,1=Mode 1, 2=Mode 2, ... 10= Random Multi Colors )
	In_LightConfigArry:	ARRAY [0..10] OF ST_LEDMode;		// Array of the color Setup
	In_AllModes_Flashing:	BYTE := 0;		// Value (Byte) for all modes to make light flash or not (0=Steady On, 1= Blinking Slow, 2= Blinking Fast) 
	
	In_ManualMode:	BOOL;	// Mode to allow LED to Run in Manual
	In_ManualValues:	ST_RGB;		// Manual RGB Values for the LED output (0=Off, 255= Full ON 100%)
		
	CFG_FlshingControl:	BOOL;	// Bit to set where blinking control comes from.  (False = In_FlashingAllModes controls all modes, TRUE = each mode is controled individually from the configuration array) 
	CFG_BlinkTimeSlowON:	TIME := T#1S;
	CFG_BlinkTimeSlowOFF:	TIME := T#500MS;
	CFG_BlinkTimeFastON:	TIME := T#500MS;
	CFG_BlinkTimeFastOFF:	TIME := T#250MS;
END_VAR
VAR_OUTPUT
	R_Out:	BYTE;	// Red LED output Byte (0=Off, 255= Full ON 100%)
	G_Out:	BYTE;	// Green LED output Byte (0=Off, 255= Full ON 100%)
	B_Out:	BYTE;	// Blue LED output Byte (0=Off, 255= Full ON 100%)
END_VAR
VAR
	PulseSlow: FB_Flasher;
	PulseFast: FB_Flasher;
	
	PulseGenerateRandom: TON;
	x: INT;
	GenerateRandom_FB: DRAND;
	RandomNumber: LREAL;
	RandomHues: ARRAY [1..3] OF BYTE;
	SlowFlashReq: BOOL;
	FastFlashReq: BOOL;
END_VAR

IF In_ManualMode THEN
	R_Out := In_ManualValues.Value_Red;
	G_Out := In_ManualValues.Value_Green;
	B_Out := In_ManualValues.Value_Blue;

ELSE
	// Set up bliking control
	SlowFlashReq := (CFG_FlshingControl AND (In_LightConfigArry[In_Light_Mode].Flashing = 1)) OR ((NOT CFG_FlshingControl) AND In_AllModes_Flashing = 1);
	FastFlashReq := (CFG_FlshingControl AND (In_LightConfigArry[In_Light_Mode].Flashing = 2)) OR ((NOT CFG_FlshingControl) AND In_AllModes_Flashing = 2);
	
	// Set Up Slow Blink Pulse If Mode is Slow Blink
	PulseSlow(In_Trig:= SlowFlashReq, Cfg_OnTime:= CFG_BlinkTimeSlowON, Cfg_OffTime:= CFG_BlinkTimeSlowOFF);

	// Set Up Fast Blink Pulse If Mode is Fast Blink
	PulseFast(In_Trig:= (FastFlashReq), Cfg_OnTime:= CFG_BlinkTimeFastON, Cfg_OffTime:= CFG_BlinkTimeFastOFF);
		
	// Set Up Random Twinkling Lights
	PulseGenerateRandom(IN:= (In_Light_Mode = 10) AND NOT PulseGenerateRandom.Q , PT:= T#250MS); 
	
	// Set Light Mode
	IF (In_Light_Mode <> 10) THEN
		IF PulseSlow.Output OR PulseFast.Output OR (CFG_FlshingControl AND In_LightConfigArry[In_Light_Mode].Flashing = 0) OR ((NOT CFG_FlshingControl) AND In_AllModes_Flashing =0) THEN
			R_Out := In_LightConfigArry[In_Light_Mode].Value1.Value_Red;
			G_Out := In_LightConfigArry[In_Light_Mode].Value1.Value_Green;
			B_Out := In_LightConfigArry[In_Light_Mode].Value1.Value_Blue;
		ELSE 
			R_Out := In_LightConfigArry[In_Light_Mode].Value2.Value_Red;
			G_Out := In_LightConfigArry[In_Light_Mode].Value2.Value_Green;
			B_Out := In_LightConfigArry[In_Light_Mode].Value2.Value_Blue;
		END_IF
	
	ELSIF In_Light_Mode = 10 THEN
		IF PulseGenerateRandom.Q THEN
			FOR x := 1 TO 3 DO
				GenerateRandom_FB(Seed:= 0, Num=> RandomNumber );
				RandomHues[x] := LREAL_TO_BYTE(RandomNumber * 255);
			END_FOR
			R_Out := RandomHues[1];
			G_Out := RandomHues[2];
			B_Out := RandomHues[3];
		END_IF
	 
	ELSE
		R_Out := 0;
		G_Out := 0;
		B_Out := 0;
	END_IF
END_IF

END_FUNCTION_BLOCK

// ---- FunctionBlocks/Metrics/FB_Metrics.TcPOU
FUNCTION_BLOCK FB_Metrics
VAR_IN_OUT
	Trigger 	: BOOL;
	HMI_Reset	: BOOL;
	TimeExpired		: BOOL;
END_VAR
VAR_INPUT
	BarcodeRead		: STRING;
END_VAR
VAR_OUTPUT
END_VAR
VAR PERSISTENT
	LoadsPassed		: DINT;
	GoodReadCount	: DINT;
	GoodReadPercent	: REAL;
	LastBarcodeRead	: STRING;
END_VAR

IF Trigger THEN	
	loadsPassed := loadsPassed + 1;	
	IF BarcodeRead <> '' THEN
		GoodReadCount := GoodReadCount + 1;
	END_IF	
	GoodReadPercent := (DINT_TO_REAL(GoodReadCount)/DINT_TO_REAL(LoadsPassed))*100;
	LastBarcodeRead := BarcodeRead;		
	Trigger := FALSE;	
END_IF

IF HMI_Reset OR TimeExpired THEN	
	LoadsPassed 		:= 0;
	GoodReadCount 		:= 0;
	GoodReadPercent		:= 0;	
	IF TimeExpired THEN	
		TimeExpired := FALSE;
	END_IF
	IF HMI_Reset THEN
		HMI_Reset := FALSE;
	END_IF
END_IF

END_FUNCTION_BLOCK

// ---- FunctionBlocks/Singulation/FB_TwoGripIndexer.TcPOU
FUNCTION_BLOCK FB_TwoGripIndexer
VAR_INPUT
	{attribute 'OPC.UA.DA' := '1'}
	In_ResetState	:	BOOL;		// Clear the current functional state of the Indexer

	In_Pause:	BOOL;
	In_ConveyorRunning			:	BOOL; //Added
	
	PE_Grabber:	BOOL;
	In_Grabber_1_Auto: BOOL;
	In_Grabber_1_Extended	:	BOOL;
	In_Grabber_1_Retracted	:	BOOL;

	
	In_SV_Grabber_1_Extend	:	BOOL;
	In_SV_Grabber_1_Retract	:	BOOL;
	
	In_EncoderCount			:	UINT;
	
	Cfg_GappingDistance		:	UINT;	// Distance in encoder Pulses before the next item can be released
	Cfg_ProductSize		    :	UINT;	// Size(length) in encoder count of product for the grabber to retract for
END_VAR
VAR_OUTPUT
	{attribute 'OPC.UA.DA' := '1'}
	Out_Homed					:	BOOL;
	{attribute 'OPC.UA.DA' := '1'}
	Out_Ready					:	BOOL;
	{attribute 'OPC.UA.DA' := '1'}
	Out_Running					:	BOOL;
	
	Out_Grabber_1_Ext:	BOOL;
	Out_Grabber_1_Ret:	BOOL;

	{attribute 'OPC.UA.DA' := '1'}
	Status:		UINT;		// General Indexer  status
	Status_Output:	UINT;	// Indexer grabber status
	
END_VAR
VAR	
	StartUp		: BOOL := TRUE;
	rPE_Grabber_1: R_TRIG;
	fPE_Grabber_1: F_TRIG;
	
	tonHomeWait					:	TON := (PT := T#1S);
	tonReadyWait				:	TON := (PT := T#1S);
	tonRunningWait				:	TON := (PT := T#5S);
	
	rResetState	:	R_TRIG;
	fRetracted	: F_TRIG; 	// Capture the Falling edge of the Induct PE
	// Extend and Retract controls
	Grabber_1_Extend		:	BOOL;
	Grabber_1_Retract		:	BOOL;
	
	RolloverDetect_HeldDist			:   UINT;
	HeldCount			    :	UINT;
	HeldDistance			:	UINT;
	RolloverDetect_ReleasedDist			:   UINT;
	ReleasedCount           :	UINT;
	ReleasedDistance        :	UINT;

	fInductPE: INT;
END_VAR

VAR CONSTANT
	// Output Status
	GRABBER_1_OCCUPIED:	UINT  := 1;
	
	// Singulation Status
	PAUSED:						UINT  := 0;
	PRODUCT_PRESENT:			UINT  := 1;
	PRODUCT_RELEASED:			UINT  := 2;
END_VAR

// Process the In_ResetState
rResetState(CLK:=In_ResetState);

IF rResetState.Q THEN
	// Clear the Status
	Status := 0;
	// Revert to the StartUp state
	StartUp := TRUE;
	// Revert to the NOT Homed state
	Out_Homed := FALSE;
	tonHomeWait(IN := FALSE);
	// Revert to the NOT Ready state
	Out_Ready := FALSE;
	tonReadyWait(IN := FALSE);
	// Revert to the NOT Running state
	Out_Running := FALSE;
	tonRunningWait(IN := FALSE);
	// Clear the reset request
	// Clear the reset request
	In_ResetState := FALSE;
END_IF

// Home the 
IF StartUp  OR NOT Out_Homed OR NOT Out_Ready THEN
	Status.PAUSED := TRUE;
	
	tonHomeWait.IN := NOT Out_Homed;
	tonHomeWait();
	IF NOT Out_Homed THEN
		// Grabber
		Grabber_1_Retract := TRUE;
		Grabber_1_Extend := FALSE;
		IF In_Grabber_1_Retracted
		   THEN
			Out_Homed := tonHomeWait.Q;
		END_IF
	END_IF

	tonReadyWait.IN := NOT Out_Ready AND Out_Homed;
	tonReadyWait();
	IF NOT Out_Ready AND Out_Homed THEN

		IF In_Grabber_1_Retracted
		   THEN
			Out_Ready := tonReadyWait.Q;
		END_IF
	END_IF

	StartUp := NOT Out_Homed OR NOT Out_Ready;
	Out_Running := FALSE;
	
ELSIF In_Pause OR NOT In_ConveyorRunning THEN
	// Grabber
	Grabber_1_Retract := TRUE;
	Grabber_1_Extend := FALSE;

ELSIF NOT Out_Running THEN
	tonRunningWait.IN := NOT OUT_Running AND Out_Ready AND Out_Homed AND In_ConveyorRunning;
	tonRunningWait();
	Out_Running := tonRunningWait.Q;

ELSIF Out_Running THEN
	Status.PAUSED := FALSE;	
		// Call Actions That run while in running state?


	END_IF
	
// Call actions???	
	
fRetracted(CLK:= In_Grabber_1_Retracted, Q =>);	
	
IF  fRetracted.Q THEN
	HeldCount := In_Encodercount;
END_IF
	
IF Releasedcount=0 AND In_Grabber_1_Retracted THEN
	ReleasedCount := In_EncoderCount;		
END_IF

IF In_Grabber_1_Retracted=0 THEN
	ReleasedCount := 0;
END_IF
	
// Singulation Distance Check, Hold for Gap
IF HeldCount <> 0 THEN
	IF In_EncoderCount > HeldCount THEN
		HeldDistance := In_EncoderCount - HeldCount;
		RolloverDetect_HeldDist := 0;
	ELSE
		// If the encoder rolls to 0, capture the last distance as an offset
		IF RolloverDetect_HeldDist = 0 THEN
			RolloverDetect_HeldDist := HeldDistance;
		END_IF
		// The new distance to check is the number of pulses from the Cleared count to the rollover (RolloverDetect)
		// 	plus the current encoder count
		HeldDistance := RolloverDetect_HeldDist + In_EncoderCount;
	END_IF
ELSE
	HeldDistance:=0;
END_IF
	
// Singulation Distance Check, release for size 
IF ReleasedCount <> 0 THEN
	IF In_EncoderCount > ReleasedCount THEN
		ReleasedDistance := In_EncoderCount - ReleasedCount;
		RolloverDetect_ReleasedDist := 0;
	ELSE
		// If the encoder rolls to 0, capture the last distance as an offset
		IF RolloverDetect_ReleasedDist = 0 THEN
			RolloverDetect_ReleasedDist := ReleasedDistance;
		END_IF
		// The new distance to check is the number of pulses from the Cleared count to the rollover (RolloverDetect)
		// 	plus the current encoder count
		ReleasedDistance  := RolloverDetect_ReleasedDist + In_EncoderCount;
	END_IF
ELSE 
	ReleasedDistance :=0;
END_IF
	
// Check Held Distance less than Gap distance
IF Cfg_GappingDistance > HeldDistance THEN
	 // Test for an item at the grabber stop
		IF PE_Grabber THEN
		//Close Grabber
		Out_Grabber_1_Ext :=TRUE;
		Out_Grabber_1_Ret :=FALSE;	
		//Reset Release count
		ELSE
		//Open Grabber
		Out_Grabber_1_Ext :=FALSE;
		Out_Grabber_1_Ret :=TRUE;
		END_IF
	//Held distance greater than Gap, Released count less than Product size 
	ELSE
		IF Cfg_ProductSize > ReleasedDistance THEN
		//Open Grabber 
		Out_Grabber_1_Ext :=FALSE;
		Out_Grabber_1_Ret :=TRUE;
		//Held distance greater than Gap, Released Greater than Product size
		ELSIF PE_Grabber THEN
		//Close Gripper
		Out_Grabber_1_Ext :=TRUE;
		Out_Grabber_1_Ret :=FALSE;
		END_IF
END_IF

	
	
	
// Activate all the outputs in one place
//Status_Output.GRABBER_1_OCCUPIED := Grabber1(Active := In_Grabber_1_Auto, Extend:= Grabber_1_Extend, Retract := Grabber_1_Retract);

END_FUNCTION_BLOCK

// ---- FunctionBlocks/Singulation/FB_TwoGripSingulation.TcPOU
FUNCTION_BLOCK FB_TwoGripSingulation
VAR_INPUT
	{attribute 'OPC.UA.DA' := '1'}
	In_ResetState	:	BOOL;		// Clear the current functional state of the Indexer

	In_Pause:	BOOL;
	In_ConveyorRunning			:	BOOL; //Added
	
	PE_Grabber:	BOOL;
	In_Grabber_1_Auto: BOOL;
	In_Grabber_1_Extended	:	BOOL;
	In_Grabber_1_Retracted	:	BOOL;
	
	In_Grabber_2_Auto: BOOL;
	In_Grabber_2_Extended	:	BOOL;
	In_Grabber_2_Retracted	:	BOOL;

	
	In_SV_Grabber_1_Extend	:	BOOL;
	In_SV_Grabber_1_Retract	:	BOOL;
	In_SV_Grabber_2_Extend	:	BOOL;
	In_SV_Grabber_2_Retract	:	BOOL;
	
	In_EncoderCount			:	UINT;
	
	Cfg_GappingDistance		:	UINT;	// Distance in encoder Pulses before the next item can be released
	Cfg_ProductSize		    :	UINT;	// Size(length) in encoder count of product for the grabber to retract for
	Cfg_GrabberSpace		:	UINT;	// Size(length) in encoder count for product to clear the grabber 
END_VAR
VAR_OUTPUT
	{attribute 'OPC.UA.DA' := '1'}
	Out_Homed					:	BOOL;
	{attribute 'OPC.UA.DA' := '1'}
	Out_Ready					:	BOOL;
	{attribute 'OPC.UA.DA' := '1'}
	Out_Running					:	BOOL;
	
	Out_Grabber_1_Ext:	BOOL;
	Out_Grabber_1_Ret:	BOOL;
	Out_Grabber_2_Ext:	BOOL;
	Out_Grabber_2_Ret:	BOOL;

	{attribute 'OPC.UA.DA' := '1'}
	Status:		UINT;		// General Indexer  status
	Status_Output:	UINT;	// Indexer grabber status
	
END_VAR
VAR	
	StartUp		: BOOL := TRUE;
	rPE_Grabber_1: R_TRIG;
	fPE_Grabber_1: F_TRIG;
	
	tonHomeWait					:	TON := (PT := T#1S);
	tonReadyWait				:	TON := (PT := T#1S);
	tonRunningWait				:	TON := (PT := T#5S);
	
	rResetState	:	R_TRIG;
	fRetracted	: F_TRIG; 	// Capture the Falling edge of the Induct PE
	// Extend and Retract controls
	Grabber_1_Extend		:	BOOL;
	Grabber_1_Retract		:	BOOL;
	Grabber_2_Extend		:	BOOL;
	Grabber_2_Retract		:	BOOL;
	
	RolloverDetect_HeldDist			:   UINT;
	HeldCount			    :	UINT;
	HeldDistance			:	UINT;
	RolloverDetect_InductDist			:   UINT;
	InductCount           :	UINT;
	InductedDistance        :	UINT;

END_VAR

VAR CONSTANT
	// Output Status
	GRABBER_1_OCCUPIED:	UINT  := 1;
	GRABBER_2_OCCUPIED:	UINT  := 2;
	
	// Singulation Status
	PAUSED:						UINT  := 0;
	PRODUCT_PRESENT:			UINT  := 1;
	PRODUCT_RELEASED:			UINT  := 2;
END_VAR

// Process the In_ResetState
rResetState(CLK:=In_ResetState);

IF rResetState.Q THEN
	// Clear the Status
	Status := 0;
	// Revert to the StartUp state
	StartUp := TRUE;
	// Revert to the NOT Homed state
	Out_Homed := FALSE;
	tonHomeWait(IN := FALSE);
	// Revert to the NOT Ready state
	Out_Ready := FALSE;
	tonReadyWait(IN := FALSE);
	// Revert to the NOT Running state
	Out_Running := FALSE;
	tonRunningWait(IN := FALSE);
	// Clear the reset request
	// Clear the reset request
	In_ResetState := FALSE;
END_IF

// Home the 
IF StartUp  OR NOT Out_Homed OR NOT Out_Ready THEN
	Status.PAUSED := TRUE;
	
	tonHomeWait.IN := NOT Out_Homed;
	tonHomeWait();
	IF NOT Out_Homed THEN
		// Grabber
		Grabber_1_Retract := TRUE;
		Grabber_1_Extend := FALSE;
		IF In_Grabber_1_Retracted
		   THEN
			Out_Homed := tonHomeWait.Q;
		END_IF
	END_IF

	tonReadyWait.IN := NOT Out_Ready AND Out_Homed;
	tonReadyWait();
	IF NOT Out_Ready AND Out_Homed THEN

		IF In_Grabber_1_Retracted
		   THEN
			Out_Ready := tonReadyWait.Q;
		END_IF
	END_IF

	StartUp := NOT Out_Homed OR NOT Out_Ready;
	Out_Running := FALSE;
	
ELSIF In_Pause OR NOT In_ConveyorRunning THEN
	// Grabber
	Grabber_1_Retract := TRUE;
	Grabber_1_Extend := FALSE;

ELSIF NOT Out_Running THEN
	tonRunningWait.IN := NOT OUT_Running AND Out_Ready AND Out_Homed AND In_ConveyorRunning;
	tonRunningWait();
	Out_Running := tonRunningWait.Q;

ELSIF Out_Running THEN
	Status.PAUSED := FALSE;	
		// Call Actions That run while in running state?


	END_IF
	
// Call actions???	
	
// HeldDistance Calculation

fRetracted(CLK:= In_Grabber_1_Retracted, Q =>);		
IF  fRetracted.Q THEN
	HeldCount := In_Encodercount;
	ELSIF In_Grabber_1_Retracted AND In_Grabber_2_Retracted THEN
	HeldCount:= 0;
END_IF
	
IF HeldCount <> 0 THEN
	IF In_EncoderCount > HeldCount THEN
	HeldDistance := In_EncoderCount - HeldCount;
	RolloverDetect_HeldDist := 0;
	ELSE
	// If the encoder rolls to 0, capture the last distance as an offset
	IF RolloverDetect_HeldDist = 0 THEN
	RolloverDetect_HeldDist := HeldDistance;
	END_IF
	// The new distance to check is the number of pulses from the Cleared count to the rollover (RolloverDetect)
	// 	plus the current encoder count
	HeldDistance := RolloverDetect_HeldDist + In_EncoderCount;
	END_IF
ELSE
	HeldDistance:=0;
END_IF

// InductedDistance Calculation

rPE_Grabber_1(CLK:= PE_Grabber, Q =>);	
IF  rPE_Grabber_1.Q THEN
	InductCount := In_Encodercount;
	ELSIF NOT PE_Grabber THEN
	InductCount := 0;	
END_IF	

// Singulation Distance Check, release for size 
IF InductCount <> 0 THEN
  IF In_EncoderCount > InductCount THEN
	InductedDistance := In_EncoderCount - InductCount;
	RolloverDetect_InductDist := 0;
	ELSE
	// If the encoder rolls to 0, capture the last distance as an offset
	IF RolloverDetect_InductDist = 0 THEN
	RolloverDetect_InductDist := InductedDistance;
		END_IF
	// The new distance to check is the number of pulses from the Cleared count to the rollover (RolloverDetect)
	// 	plus the current encoder count
	InductedDistance  := RolloverDetect_InductDist + In_EncoderCount;
	END_IF
ELSE
	InductedDistance:=0;
END_IF

 
// Grabber Motion
IF HeldDistance < Cfg_GappingDistance THEN
	IF InductedDistance > Cfg_ProductSize THEN
		Out_Grabber_1_Ext:= TRUE;
		Out_Grabber_2_Ext:= TRUE;
	ELSE
		Out_Grabber_1_Ext:= FALSE;
		Out_Grabber_2_Ext:= FALSE;
	END_IF
ELSIF HeldDistance < (Cfg_GappingDistance + Cfg_GrabberSpace) THEN
	Out_Grabber_1_Ext:= FALSE;
	Out_Grabber_2_Ext:= TRUE;
ELSE
	Out_Grabber_1_Ext:= FALSE;
	Out_Grabber_2_Ext:= FALSE;
	//HeldCount:= 0;
END_IF
		
// Activate all the outputs in one place
//Status_Output.GRABBER_1_OCCUPIED := Grabber1(Active := In_Grabber_1_Auto, Extend:= Grabber_1_Extend, Retract := Grabber_1_Retract);

END_FUNCTION_BLOCK

// ---- FunctionBlocks/Sorter/ProcessBuffers.TcPOU
PROGRAM ProcessBuffers
VAR_IN_OUT
	st_NextToInduct					: ST_ItemTemporary;
	st_UpdateItem					: ST_ItemTemporary;
	st_TempInductItem				: ST_ItemTemporary;
	st_Sorter						: ST_Sorter;
	aDiverts						: ARRAY[SorterExample.DIVERTMIN..SorterExample.NUMBEROFDIVERTS] OF ST_DIVERT;
	aItems 							: ARRAY[SorterExample.SORTERENCODERMIN..SorterExample.SORTERENCODERMAX] OF ST_Item;
END_VAR

VAR_INPUT
	DivertToCommission				: DINT;
	ItemsArrayMax 					: UDINT;
	ItemsArrayMin 					: UDINT;
END_VAR
VAR
	st_ArrivalBuffer AT %I* 		: ST_ItemBuffer;
	st_ArrivalFdbkIn				: ST_ItemBufferFdbk;
	st_ArrivalFdbkOut	AT %Q*		: ST_ItemBufferFdbk;
	fb_ArrivalBuffer				: FB_ItemBuffer;
	st_ArrivalItem 					: ST_Item;		// Arrival Item (Bar code read) from System PLC (BarCodeReaders.pou)

	// Item to replace in the sorter buffer
	st_ReplaceItem					: st_Item;

	st_TransportBuffer AT %I* 		: ST_ItemBuffer;
	st_TransportFdbkIn				: ST_ItemBufferFdbk;
	st_TransportFdbkOut	AT %Q*		: ST_ItemBufferFdbk;
	fb_TransportBuffer				: FB_ItemBuffer;

	st_UpdateBuffer AT %Q* 			: ST_ItemBuffer;
	st_UpdateFdbkIn	AT %I*			: ST_ItemBufferFdbk;
	st_UpdateFdbkOut				: ST_ItemBufferFdbk;
	fb_UpdateBuffer 				: FB_ItemBuffer;

	st_ToUpdate						: ST_ItemTemporary;	// Item to Update on the Sorter, or waiting to be added to the sorter

	ItemsArraySize			: UDINT;

	TransportItemInSorter	: ST_Item;	// Temporary Processing Item
	TransportItemFound		: ST_Item;	// Item to Update Found
	TransportSorterIndex	: UDINT;

	ExitSorterIndex			: UDINT;
	ExitItemInSorter		: ST_Item;
	ExitItemFound			: ST_ItemTemporary;
	ExitInDivert			: BOOL;
	ExitDiverting			: BOOL;
	ExitSuccess				: BOOL;
	ExitDetected			: BOOL;
	ExitComplete			: BOOL;

	UpdateIndexCounter		: DINT;

	bTest : BOOL;
	sMessage	:	STRING;
	
	st_DisplayItem		:st_Item;
	LogSorterDump		:BOOL := FALSE;
	aTestBool			:	ARRAY[0..100] OF BOOL;
	
	fb_FindDestination		: FB_FindDestination;
	fb_DefaultDestination	: FB_FindDestination;
	fb_RecircDestination	: FB_FindDestination;
	// Created to allow the aDiverts to be used in the FB_FindDestination Function Block
	aTempDiverts			: ARRAY[SorterExample.DIVERTMIN..SorterExample.NUMBEROFDIVERTS] OF ST_DIVERT;
END_VAR


aTempDiverts := aDiverts;
// Initialize the Transport and Update buffers
// Set Master for FB's that control the buffer
fb_ArrivalBuffer.Master := FALSE;
fb_TransportBuffer.Master := FALSE;
fb_UpdateBuffer.Master := TRUE;

// Turn ON/OFF Logging of all activity in/out
fb_ArrivalBuffer.LogEntries := .nItemBufferLogEnable.ARRIVALS;
fb_TransportBuffer.LogEntries := .nItemBufferLogEnable.TRANSPORT;
fb_UpdateBuffer.LogEntries := .nItemBufferLogEnable.UPDATE;

// Provide names for the buffers
fb_ArrivalBuffer.Name := 'SRT ARRIVAL';
fb_TransportBuffer.Name := 'SRT TRANSPORT';
fb_UpdateBuffer.Name := 'SRT UPDATE';

// Initialize the FB_ItemExtBuffer Instances
fb_ArrivalBuffer(st_BufferData := st_ArrivalBuffer
						, st_BufferFdbkIn := st_ArrivalFdbkIn
						, st_BufferFdbkOut => st_ArrivalFdbkOut);
fb_TransportBuffer(st_BufferData := st_TransportBuffer
						, st_BufferFdbkIn := st_TransportFdbkIn
						, st_BufferFdbkOut => st_TransportFdbkOut);
fb_UpdateBuffer(st_BufferData := st_UpdateBuffer
						, st_BufferFdbkIn := st_UpdateFdbkIn
						, st_BufferFdbkOut => st_UpdateFdbkOut);

IF GVL_IO.INIT THEN
	fb_ArrivalBuffer.Clear();
	fb_TransportBuffer.Clear();
	fb_UpdateBuffer.Clear();
END_IF
						
(*
	Set the Upper/Lower bound of relevant arrays for looping purposes
	ItemsArrayMax/Min for the sorter array slot count
*)
// Size is Max - Min + 1 to capture both extremes
ItemsArraySize := ItemsArrayMax - ItemsArrayMin + 1;

(*
 	Check for a value disagreement in the Arrival Buffer In and Out pointers to
  	determine if there is an update for an item.
	When an Item arrives, the System PLC adds it to the shared buffer and increments
	the InPointer
*)
IF st_ArrivalBuffer.nInPointer <> fb_ArrivalBuffer.OutPointer THEN
	fb_ArrivalBuffer.RemoveItem(st_ItemToReturn => st_ArrivalItem);
END_IF

// Input Item read at bar code reader from System PLC to sorter
IF st_ArrivalItem.ID <> '' THEN
	IF .nSortBufferLogEnable.BUFFER_ARRIVAL THEN
		sMessage := CONCAT(' Item: ', st_ArrivalItem.ID);
		sMessage := CONCAT(sMessage,' Pulses: ');
		sMessage := CONCAT(sMessage, UDINT_TO_STRING(st_Sorter.EncoderCounts));
		// Write to the Error List
		ADSLOGSTR( msgCtrlMask := ADSLOG_MSGTYPE_HINT OR ADSLOG_MSGTYPE_LOG
			, msgFmtStr := 'Arrival Processed: %s'
			, strArg := sMessage);
	END_IF
	// Indicate that this item did not get added to the sorter and add to the exit buffer
	//  Both as a TransportUpdate and TransportComplete message type 
	IF st_NextToInduct.Item.ID <> '' THEN
		IF .nSortBufferLogEnable.BUFFER_MISSINDUCT THEN
			sMessage := CONCAT(' Item: ', st_NextToInduct.Item.ID);
			// Write to the Error List
			ADSLOGSTR( msgCtrlMask := ADSLOG_MSGTYPE_HINT OR ADSLOG_MSGTYPE_LOG
				, msgFmtStr := 'Item Removed - Not Inducted: %s'
				, strArg := sMessage);
		END_IF
		// Transport Response
		st_NextToInduct.Item.Status := E_StatusCode.Assign_NotInducted;
		st_NextToInduct.Item.DeviceID := st_Sorter.Config.EquipID;
		st_NextToInduct.Item.MessageType := E_MessageIds.TransportResponse_25;
		fb_UpdateBuffer.AddItem(st_ItemToAdd := st_NextToInduct.Item);

		// Transport Complete
		st_NextToInduct.Item.Status := E_StatusCode.Divert_NotInducted;
		st_NextToInduct.Item.MessageType := E_MessageIds.TransportComplete_26;
		fb_UpdateBuffer.AddItem(st_ItemToAdd := st_NextToInduct.Item);
	END_IF
	// Copy Last BCR item to Item to Induct
	st_NextToInduct.Item :=  st_ArrivalItem;
	// Add the Sorter EquipID to the NextToInduct
	st_NextToInduct.Item.DeviceID := st_Sorter.Config.EquipID;
	// Set the Default Destination
	st_NextToInduct.Item.Destination := st_Sorter.Config.DefaultDestination;
	// Capture an encoder value that when the encoder count exceeds this value, NextToInduct item will be cleared
	st_NextToInduct.Counts := st_Sorter.EncoderCounts;
	// Clear the Last recieved item
	st_ArrivalItem := BlankItem;
	// Prepare to replace the Temporarily assigned item with this item
	IF st_TempInductItem.Item.ID <> '' THEN
		// Capture the Counts and Length from the temporary item
		st_NextToInduct.Counts := st_TempInductItem.Counts;
		st_NextToInduct.Item.Length := st_TempInductItem.Item.Length;
		//Identify the Item to replace in the sorter array
		st_ReplaceItem := st_TempInductItem.Item;
		st_TempInductItem.Counts := 0;
		st_TempInductItem.Item := BlankItem;
		IF .nSortBufferLogEnable.BUFFER_TEMPINDUCT THEN
			ADSLOGSTR( msgCtrlMask := ADSLOG_MSGTYPE_HINT OR ADSLOG_MSGTYPE_LOG
				, msgFmtStr := 'Temp ID Replaced : %s'
				, strArg := st_ReplaceItem.ID); 
		END_IF
	END_IF
END_IF

(*
 	Check for a value disagreement in the SorterTransportBuffer In and Out pointers to
  	determine if there is an update for an item.
	When an update arrived, the System PLC adds it to the shared buffer and increments
	the InPointer
*)
IF st_TransportBuffer.nInPointer <> fb_TransportBuffer.OutPointer THEN
	fb_TransportBuffer.RemoveItem(st_ItemToReturn => st_ToUpdate.Item);
	// Lookup the index for the chosen destination
	fb_FindDestination(RoundRobin := st_Sorter.Config.RoundRobin
					, aDiverts := aTempDiverts
					, DestinationID := st_ToUpdate.Item.Destination
					, DestinationIndex => st_ToUpdate.Item.DestinationIdx);
	IF .nSortBufferLogEnable.BUFFER_DESTINDEX THEN
		sMessage := CONCAT(' Item: ', st_ToUpdate.Item.ID);
		sMessage := CONCAT(sMessage,' Destination: ');
		sMessage := CONCAT(sMessage, UDINT_TO_STRING(TransportSorterIndex));
		sMessage := CONCAT(sMessage,' Index: ');
		sMessage := CONCAT(sMessage, UDINT_TO_STRING(TransportSorterIndex));
		// Write to the Error List
		ADSLOGSTR( msgCtrlMask := ADSLOG_MSGTYPE_HINT OR ADSLOG_MSGTYPE_LOG
			, msgFmtStr := 'Divert Index of Destination: %s'
			, strArg := sMessage);
	END_IF
END_IF

// Get the Default Destination Index
fb_DefaultDestination(RoundRobin := st_Sorter.Config.RoundRobin
				, aDiverts := aTempDiverts
				, DestinationID := st_Sorter.Config.DefaultDestination
				, DestinationIndex => st_Sorter.Config.DefaultDestIdx);

// Get the Recirculation Destination Index
fb_RecircDestination(RoundRobin := st_Sorter.Config.RoundRobin
				, aDiverts := aTempDiverts
				, DestinationID := st_Sorter.Config.RecircDestination
				, DestinationIndex => st_Sorter.Config.RecircDestIdx);

// Test the Item to Update against the Item to Induct and update if they match:
//	Update the NextItemToInduct with the updated data, then clear the Item to Update
IF st_ToUpdate.Item.ID <> '' THEN
	IF st_ToUpdate.Item.ID = st_NextToInduct.Item.ID THEN
		// Indicate that the transport command was received and a response was sent
		st_NextToInduct.Item.MessageType := E_MessageIds.TransportResponse_25;
		// Test the assigned lane for availability
		IF aDiverts[st_ToUpdate.Item.DestinationIdx].Full
		   OR aDiverts[st_ToUpdate.Item.DestinationIdx].Faulted THEN
			// Prepare a message to indicate that the item cannot be assigned
			st_ToUpdate.Item.Status := E_StatusCode.Assign_Full;
			st_ToUpdate.Item.DeviceID := st_Sorter.Config.EquipID;
			st_ToUpdate.Item.MessageType := E_MessageIds.TransportResponse_25;
			fb_UpdateBuffer.AddItem(st_ItemToAdd := st_ToUpdate.Item);
			st_NextToInduct.Item.ExtStatus := E_StatusCode.Divert_Full;
		ELSE
			st_NextToInduct.Item.DeviceID := st_Sorter.Config.EquipID;
			st_NextToInduct.Item.Status := E_StatusCode.Assign_Accepted;
			// Update the Destination
			st_NextToInduct.Item.Destination := st_ToUpdate.Item.Destination;
			st_NextToInduct.Item.DestinationIdx := st_ToUpdate.Item.DestinationIdx;
			fb_UpdateBuffer.AddItem(st_ItemToAdd := st_NextToInduct.Item);
		END_IF
		// If commissioning, ignore any other direction
		IF DivertToCommission > 0 THEN
			st_NextToInduct.Item.Destination := DivertToCommission;
		END_IF
		// Log the update
		IF .nSortBufferLogEnable.BUFFER_INDUCT THEN
			sMessage := CONCAT(' Item: ', st_ToUpdate.Item.ID);
			sMessage := CONCAT(sMessage,' Pulses: ');
			sMessage := CONCAT(sMessage, UDINT_TO_STRING(st_Sorter.EncoderCounts));
			sMessage := CONCAT(sMessage,' Status: ');
			sMessage := CONCAT(sMessage, UDINT_TO_STRING(st_ToUpdate.Item.Status));
			sMessage := CONCAT(sMessage,' Ext Status: ');
			sMessage := CONCAT(sMessage, UDINT_TO_STRING(st_ToUpdate.Item.ExtStatus));
			// Write to the Error List
			ADSLOGSTR( msgCtrlMask := ADSLOG_MSGTYPE_HINT OR ADSLOG_MSGTYPE_LOG
				, msgFmtStr := 'Found Before Induct: %s'
				, strArg := sMessage);
		END_IF
		// We updated the item we were inducting, clear the Item to update
		st_ToUpdate.Item := BlankItem;
	END_IF
END_IF

// Clear the Update Item Found record each pass
TransportItemFound := BlankItem;

// Clear the last detected Exit item
ExitItemFound.Item := BlankItem;

// Reset the Detection booleans
ExitInDivert := FALSE;
ExitDiverting := FALSE;
ExitDetected := FALSE;
ExitSuccess := FALSE;
ExitComplete := FALSE;

// Loop through the entire array, it should be appropriately sized for the length of the sorter section
FOR UpdateIndexCounter := UDINT_TO_DINT(ItemsArrayMin) TO UDINT_TO_DINT(ItemsArrayMax) DO //Loop through everything in the sorter	

	// For Transport commands, start from the current encoder count and work forwards, just like the exit
	TransportSorterIndex := F_CalculateIndex(Offset := (UpdateIndexCounter)
											, InitialValue := st_Sorter.EncoderCounts
											, BufferSize := ItemsArraySize);

	// This is the item in the sorter array that we will be procesing this pass, testing for a Transport update message
	TransportItemInSorter := aItems[UDINT_TO_DINT(TransportSorterIndex)];

	// Test for a replace item
	// ReplaceItem is the temporary item
	// NextToInduct is the item to replace the temporary with
	IF st_ReplaceItem.ID <> '' THEN
		IF st_ReplaceItem.ID = TransportItemInSorter.ID THEN
			IF .nSortBufferLogEnable.BUFFER_REPLACEINDUCT THEN
				sMessage := CONCAT(' Item: ', st_ReplaceItem.ID);
				sMessage := CONCAT(sMessage,' New Item: ');
				sMessage := CONCAT(sMessage, st_NextToInduct.Item.ID);
				sMessage := CONCAT(sMessage,' Index: ');
				sMessage := CONCAT(sMessage, UDINT_TO_STRING(TransportSorterIndex));
				sMessage := CONCAT(sMessage,' Orig Dest: ');
				sMessage := CONCAT(sMessage, DINT_TO_STRING(TransportItemInSorter.Destination));
				sMessage := CONCAT(sMessage,' New Dest: ');
				sMessage := CONCAT(sMEssage, DINT_TO_STRING(st_ReplaceItem.Destination));
				// Write to the Error List
				ADSLOGSTR( msgCtrlMask := ADSLOG_MSGTYPE_HINT OR ADSLOG_MSGTYPE_LOG
					, msgFmtStr := 'Item ID Replaced After Induct: %s'
					, strArg := sMessage);
			END_IF
			TransportItemInSorter.ID := st_NextToInduct.Item.ID;
			TransportItemInSorter.Destination := st_NextToInduct.Item.Destination;
			TransportItemInSorter.DeviceID := st_NextToInduct.Item.DeviceID;
			TransportItemInSorter.MessageType := st_NextToInduct.Item.MessageType;
			TransportItemInSorter.Status := st_NextToInduct.Item.Status;
			TransportItemInSorter.UniqueID := st_NextToInduct.Item.UniqueID;
			TransportItemInSorter.CapturedInMetrics := st_NextToInduct.Item.CapturedInMetrics;
		END_IF
	END_IF
	// Test for an Item Update
	IF st_ToUpdate.Item.ID <> '' THEN
		// Test the sorter item against the update item
		IF st_ToUpdate.Item.ID = TransportItemInSorter.ID THEN
			IF .nSortBufferLogEnable.BUFFER_UPDATEINDUCT THEN
				sMessage := CONCAT(' Item: ', st_ToUpdate.Item.ID);
				sMessage := CONCAT(sMessage,' Index: ');
				sMessage := CONCAT(sMessage, UDINT_TO_STRING(TransportSorterIndex));
				// Write to the Error List
				ADSLOGSTR( msgCtrlMask := ADSLOG_MSGTYPE_HINT OR ADSLOG_MSGTYPE_LOG
					, msgFmtStr := 'Found After Induct: %s'
					, strArg := sMessage);
			END_IF
			// Copy the found item record, 
			TransportItemFound := TransportItemInSorter;
			// Test the destined divert for availability
			IF aDiverts[st_ToUpdate.Item.DestinationIdx].Full OR aDiverts[st_ToUpdate.Item.DestinationIdx].Faulted THEN
				// Prepare a message to indicate that the item cannot be assigned
				TransportItemFound.Status := E_StatusCode.Assign_Full;
				TransportItemFound.ExtStatus := E_StatusCode.Divert_Full;
				TransportItemFound.MessageType := E_MessageIds.TransportResponse_25;
				TransportItemFound.Destination := st_Sorter.Config.DefaultDestination;
				TransportItemFound.DestinationIdx := st_Sorter.Config.DefaultDestIdx;
			// Test for an already diverting item and assign an ExtStatus of LateAssignment
			ELSIF TransportItemInSorter.Status >= E_StatusCode.Diverting THEN
				TransportItemFound.ExtStatus := E_StatusCode.Divert_LateAssignment;
				TransportItemFound.MessageType := E_MessageIds.TransportResponse_25;
			ELSE
				//  Change the destination, which should be the only item in the update
				TransportItemFound.Destination := st_ToUpdate.Item.Destination;
				TransportItemFound.DestinationIdx := st_ToUpdate.Item.DestinationIdx;
				// This message indicates we could assign the Item
				TransportItemFound.Status := E_StatusCode.Assign_Accepted;
				TransportItemFound.MessageType := E_MessageIds.TransportResponse_25;
			END_IF
			TransportItemFound.DeviceID := st_Sorter.Config.EquipID;
			// Add the item to the update buffer
			fb_UpdateBuffer.AddItem(TransportItemFound);
			// Clear the ToUpdate Item
			st_ToUpdate.Item := BlankItem;
		END_IF
	END_IF
	
	IF TransportItemFound.ID <> '' THEN
		// Test the sorter item against the update item
		IF TransportItemFound.ID = TransportItemInSorter.ID THEN
			// Only update if it is different
			IF TransportItemFound.Destination <> TransportItemInSorter.Destination THEN
				IF .nSortBufferLogEnable.BUFFER_UPDATEDEST THEN
					sMessage := CONCAT(' Item: ', TransportItemInSorter.ID);
					sMessage := CONCAT(sMessage,' Index: ');
					sMessage := CONCAT(sMessage, UDINT_TO_STRING(TransportSorterIndex));
					sMessage := CONCAT(sMessage,' Orig Dest: ');
					sMessage := CONCAT(sMessage, DINT_TO_STRING(TransportItemInSorter.Destination));
					sMessage := CONCAT(sMessage,' Orig DeviceID ');
					sMessage := CONCAT(sMessage, TransportItemInSorter.DeviceID);
					// Write to the Error List
					ADSLOGSTR( msgCtrlMask := ADSLOG_MSGTYPE_HINT OR ADSLOG_MSGTYPE_LOG
						, msgFmtStr := 'Dest Updated After Induct: %s'
						, strArg := sMessage);
				END_IF
				// Update the Destination. If the destination is unavailable, it has been already been set to the default
				TransportItemInSorter.Destination := TransportItemFound.Destination;
				TransportItemInSorter.DeviceID := TransportItemFound.DeviceID;
				TransportItemInSorter.MessageType := TransportItemFound.MessageType;
				TransportItemInSorter.Status := TransportItemFound.Status;
				TransportItemInSorter.ExtStatus := TransportItemFound.ExtStatus;
	
				IF .nSortBufferLogEnable.BUFFER_UPDATEDEST THEN
					sMessage := CONCAT(' Item: ', TransportItemInSorter.ID);
					sMessage := CONCAT(sMessage,' Index: ');
					sMessage := CONCAT(sMessage, UDINT_TO_STRING(TransportSorterIndex));
					sMessage := CONCAT(sMessage,' New Dest: ');
					sMessage := CONCAT(sMessage, DINT_TO_STRING(TransportItemInSorter.Destination));
					sMessage := CONCAT(sMessage,' New DeviceID ');
					sMessage := CONCAT(sMessage, TransportItemInSorter.DeviceID);
					// Write to the Error List
					ADSLOGSTR( msgCtrlMask := ADSLOG_MSGTYPE_HINT OR ADSLOG_MSGTYPE_LOG
						, msgFmtStr := 'Dest Updated After Induct: %s'
						, strArg := sMessage);
				END_IF
			END_IF
			// Make sure that the destination update makes it to the item being inducted into the sorter
			IF st_UpdateItem.Item.ID <> '' THEN
				IF st_UpdateItem.Item.ID = TransportItemFound.ID THEN
					IF st_UpdateItem.Item.Destination <> TransportItemFound.Destination THEN
						IF .nSortBufferLogEnable.BUFFER_UPDATEDEST THEN
							// Log the original destination
							sMessage := CONCAT(' Item: ', st_UpdateItem.Item.ID);
							sMessage := CONCAT(sMessage, ' Pulses: ');
							sMessage := CONCAT(sMessage, UDINT_TO_STRING(st_Sorter.EncoderCounts));
							sMessage := CONCAT(sMessage,' Orig Dest: ');
							sMessage := CONCAT(sMessage, DINT_TO_STRING(st_UpdateItem.Item.Destination));
							// Write to the Error List
							ADSLOGSTR( msgCtrlMask := ADSLOG_MSGTYPE_HINT OR ADSLOG_MSGTYPE_LOG
								, msgFmtStr := 'Induct Dest Changed: %s'
								, strArg := sMessage);
						END_IF
						// Update the Destination
						st_UpdateItem.Item.Destination := TransportItemFound.Destination;
						// Log the new destination
						IF .nSortBufferLogEnable.BUFFER_UPDATEDEST THEN
							sMessage := CONCAT(' Item: ', st_UpdateItem.Item.ID);
							sMessage := CONCAT(sMessage, ' Pulses: ');
							sMessage := CONCAT(sMessage, UDINT_TO_STRING(st_Sorter.EncoderCounts));
							sMessage := CONCAT(sMessage,' New Dest: ');
							sMessage := CONCAT(sMessage, DINT_TO_STRING(st_UpdateItem.Item.Destination));
							// Write to the Error List
							ADSLOGSTR( msgCtrlMask := ADSLOG_MSGTYPE_HINT OR ADSLOG_MSGTYPE_LOG
								, msgFmtStr := 'Induct Dest Changed: %s'
								, strArg := sMessage);
						END_IF
					END_IF
				END_IF
			ELSE
				IF .nSortBufferLogEnable.BUFFER_UPDATEDEST THEN
					sMessage := CONCAT(' Item: ', TransportItemInSorter.ID);
					sMessage := CONCAT(sMessage,' Index: ');
					sMessage := CONCAT(sMessage, UDINT_TO_STRING(TransportSorterIndex));
					sMessage := CONCAT(sMessage,' Orig Dest: ');
					sMessage := CONCAT(sMessage, DINT_TO_STRING(TransportItemInSorter.Destination));
					// Write to the Error List
					ADSLOGSTR( msgCtrlMask := ADSLOG_MSGTYPE_HINT OR ADSLOG_MSGTYPE_LOG
						, msgFmtStr := 'Dest Received After Induct: %s'
						, strArg := sMessage);
				END_IF
				
			END_IF
		END_IF
	END_IF

	// Put the updated record back into the array
	aItems[TransportSorterIndex] := TransportItemInSorter;
	
//==================================================
// 	Done procesing Transport information
//
//	Begin processing Update/Exit information
//==================================================
	
	// For exits, start from the current encoder count and work forward
	ExitSorterIndex := F_CalculateIndex(Offset := UpdateIndexCounter
										, InitialValue := st_Sorter.EncoderCounts
										, BufferSize := ItemsArraySize);

	// Identify the Item we are testing
	ExitItemInSorter := aItems[ExitSorterIndex];

	// Populated ID identifies an item in the sorter
	// Between the two Divert status codes indicates that the item has attempted to divert
	IF ExitItemInSorter.ID <> '' THEN
		// Capture the Item encoder index and the Item at the current index
		//  This represents the first item record for this item
		//  It is captured to log the start index to allow this first record to be updated
		//  when the item is completely diverted
		IF ExitItemFound.Item.ID = '' THEN
			ExitItemFound.Counts := ExitSorterIndex;
			ExitItemFound.Item := ExitItemInSorter;
			IF ExitItemFound.Item.Status = E_StatusCode.Divert_Complete THEN
				ExitComplete := TRUE;
			END_IF
		END_IF
		// When ExitComplete is TRUE, and the ID's match, clear out this Item
		IF ExitComplete THEN
			IF ExitItemInSorter.ID = ExitItemFound.Item.ID THEN
				IF aItems[ExitSorterIndex].ID <> '' THEN
					IF .nSortBufferLogEnable.BUFFER_DUMP THEN
						sMessage := CONCAT(' Item: ', aItems[ExitSorterIndex].ID);
						sMessage := CONCAT(sMessage,' Index: ');
						sMessage := CONCAT(sMessage, UDINT_TO_STRING(ExitSorterIndex));
						sMessage := CONCAT(sMessage,' Item Status: ');
						sMessage := CONCAT(sMessage, DINT_TO_STRING(aItems[ExitSorterIndex].Status));
						sMessage := CONCAT(sMessage,' Item Ext Status: ');
						sMessage := CONCAT(sMessage, DINT_TO_STRING(aItems[ExitSorterIndex].ExtStatus));
						// Write to the Error List
						ADSLOGSTR( msgCtrlMask := ADSLOG_MSGTYPE_HINT OR ADSLOG_MSGTYPE_LOG
							, msgFmtStr := 'Exit Complete Dump Info: %s'
							, strArg := sMessage);
					END_IF
				END_IF
				aItems[ExitSorterIndex] := BlankItem;
			END_IF
		// When ExitComplete is FALSE, test for a diverting/diverted item
		ELSE
			// Detect when this item is in a diverting state
			IF (ExitItemInSorter.Status >= E_StatusCode.Diverting
			   OR ExitItemInSorter.Status <= E_StatusCode.Divert_Success)
			   THEN
			   	ExitInDivert := TRUE;
				(*
					Status value increase from Diverting to Divert_Complete
					Codes to indicate divert disposition are between Diverting and Divert_Detected
					Divert_Full and Diverting are set in FB_DivertDecision/FB_DivertControl
					Divert_Detected, Divert_Success, and Divert_Missed are set in FB_ConfirmCheck
				*)
				ExitDiverting := TRUE;
				IF ExitItemInSorter.Status = E_StatusCode.Divert_Detected THEN
					ExitDetected := TRUE;
				END_IF
				// Once the divert is successful, we are no longer "diverting"
				IF ExitItemInSorter.Status = E_StatusCode.Divert_Success THEN
					ExitSuccess := TRUE;
					ExitDiverting := FALSE;
				END_IF
				(*	
					ExitItemInSorter is the current item being examined
					ExitItemFound.Item is a copy of the Array item at ExitItemFound.Counts
					ExitItemFound.Counts references the Array index of the first record associated with this item
					When a Status/ExtStatus of greater value is detected, the first record Status/ExtStatus is overwritten
					The ExitItemFound.Item.Status/.ExtStatus is also updated
				*)
				IF ExitItemInSorter.Status > aItems[ExitItemFound.Counts].Status THEN
					aItems[ExitItemFound.Counts].Status := ExitItemInSorter.Status;
					ExitItemFound.Item.Status := ExitItemInSorter.Status;
				END_IF
				IF ExitItemInSorter.ExtStatus > aItems[ExitItemFound.Counts].ExtStatus THEN
					aItems[ExitItemFound.Counts].ExtStatus := ExitItemInSorter.ExtStatus;
					ExitItemFound.Item.ExtStatus := ExitItemInSorter.ExtStatus;
				END_IF
			END_IF
			aItems[ExitSorterIndex].Status := ExitItemFound.Item.Status;
		END_IF
	ELSE
		(*
			This path is followed when the ExitItemInSorter.ID is empty, which indicates
			that the array record associated with this index is not occupied

			ExitInDivert, ExitDiverting and ExitSuccess are all set while the .ID is not empty
		*)
		// This item was in a "diverting" state
		IF ExitInDivert THEN
			// This item is not currently diverting
			IF NOT ExitDiverting THEN
				// Only change to a Divert_Success if a Divert_Success was detected
				// Any other status is captured in the ELSE clause of the CASE statement
				IF ExitSuccess THEN
					ExitItemFound.Item.Status := E_StatusCode.Divert_Success;
				END_IF
				ExitItemFound.Item.CapturedInMetrics := TRUE;
				ExitItemFound.Item.MessageType := E_MessageIds.TransportComplete_26;
				fb_UpdateBuffer.AddItem(ExitItemFound.Item);
				aItems[ExitItemFound.Counts].Status := E_StatusCode.Divert_Complete;
			END_IF
		END_IF
		// Clear the last detected Exit item
		ExitItemFound.Item := BlankItem;
		// Reset the Detection booleans
		ExitInDivert := FALSE;
		ExitDiverting := FALSE;
		ExitDetected := FALSE;
		ExitSuccess := FALSE;
		ExitComplete := FALSE;
	END_IF
END_FOR

// If the ID is populated, we didn't find a match to update
IF st_ToUpdate.Item.ID <> '' THEN
	IF .nSortBufferLogEnable.BUFFER_UNASSIGNED THEN
		sMessage := CONCAT(' Item: ', st_ToUpdate.Item.ID);
		// Write to the Error List
		ADSLOGSTR( msgCtrlMask := ADSLOG_MSGTYPE_HINT OR ADSLOG_MSGTYPE_LOG
			, msgFmtStr := 'Item Not Updated: %s'
			, strArg := sMessage);
	END_IF
	st_ToUpdate.Item.Status := E_StatusCode.Assign_NotFound;
	st_ToUpdate.Item.DeviceID := st_Sorter.Config.Name;
	st_ToUpdate.Item.MessageType := E_MessageIds.TransportResponse_25;
	fb_UpDateBuffer.AddItem(st_ItemToAdd := st_ToUpdate.Item);
	st_ToUpdate.Item := BlankItem;
END_IF

END_PROGRAM

// ---- FunctionBlocks/Sorter/SorterExample.TcPOU
PROGRAM SorterExample
VAR
	nSorterClearIdx				: DINT;
	bSimulate					: BOOL := FALSE;	// Indicates when runing a simulation
	BlankItem					: ST_Item := (ID := ''
												, UniqueID := 0
												, Destination := 0
												, Status := E_StatusCode.No_Status
												, ExtStatus := E_StatusCode.No_Status
												, DeviceID := ''
												, MessageType := E_MessageIds.NoMessage_00);
	
	st_ToInduct					: ST_ItemTemporary;	// This is the next item to be inducted onto the sorter
	st_Inducting				: ST_ItemTemporary;	// This is the next item to be inducted onto the sorter
	st_InductUpdate				: ST_ItemTemporary;	// This is to update an item already being inducted
	{attribute 'OPC.UA.DA' := '1'}
	st_Sorter					: ST_Sorter;
	{attribute 'OPC.UA.DA' := '1'}
	aSorterDiverts 				: ARRAY[DIVERTMIN..NUMBEROFDIVERTS] OF ST_Divert;

	st_SorterEncoder 			: ST_Encoder;
	fb_SorterEncoder 			: FB_ProcessEncoder;
	{attribute 'OPC.UA.DA' := '1'}
	ENC_Raw	AT %I*:	UINT;	// Raw Encoder Value
	tEncoderOK			: TON;
	nLastEncoderCount	: UDINT;

	{attribute 'OPC.UA.DA' := '1'}
	fb_SortMetrics				: FB_Metrics;

	In_DefaultDestination AT %I*	: DINT;	// Input default destination update from Host messaging(MsgControl.RECEIVE)

	fb_CommissionSorterDiverts	: FB_DivertCommission;
	rInductPE					: R_TRIG; 	// Capture the Rising edge of the Induct PE
	fInductPE					: F_TRIG; 	// Capture the Falling edge of the Induct PE

	rDischargePE				: R_TRIG; 	// Capture the Rising edge of the Discharge PE
	fDischargePE				: F_TRIG; 	// Capture the Falling edge of the Discharge PE

	st_TempItem					: ST_ItemTemporary;	// Store temporary Item info until BCR data is received

	DivertToCommission			: UINT := 0;	// Non-zero value will send all items to this divert

	sMessage			: STRING;

	ClearSorterArray	: BOOL;

	FB_DivertLog		: FB_DivertLog;
	
	SorterDischargeItem	: ST_Item;

END_VAR

VAR PERSISTENT
	aSorterItems 				: ARRAY[SORTERENCODERMIN..SORTERENCODERMAX] OF ST_Item;	// Persist the Items to Sort array
	{attribute 'OPC.UA.DA' := '1'}
	st_SorterCfg				: ST_SorterConfig; 	// Persist Sorter configuration
	{attribute 'OPC.UA.DA' := '1'}
	aSorterDivertsCfgs 			: ARRAY[DIVERTMIN..NUMBEROFDIVERTS] OF ST_DivertCfg; 	// Persist Sorter Configuration
END_VAR

VAR CONSTANT
	SORTERMASKSIZE				: UINT := 11;		// Number of bits to mask into the Encoder Count, will define the size of the SORTERENCODERMAX value
	{attribute 'OPC.UA.DA' := '1'}
	NUMBEROFDIVERTS				: DINT := 3;
	DIVERTMIN					: DINT := 1;
	{attribute 'OPC.UA.DA' := '1'}
	SORTERENCODERMAX			: UDINT := ((LREAL_TO_UDINT(EXPT(2,SORTERMASKSIZE)))-1); // Calculated size based on the bitmask 
	{attribute 'OPC.UA.DA' := '1'}
	SORTERENCODERMIN			: UDINT := 0;

END_VAR

// Sorter clear when the system is restarted or downloaded (INIT=TRUE for first scan)
IF (GVL_IO.INIT AND NOT st_SorterCfg.RetainOnRestart) OR ClearSorterArray THEN
	FOR nSorterClearIdx := UDINT_TO_DINT(SORTERENCODERMIN) TO UDINT_TO_DINT(SORTERENCODERMAX) BY 1 DO
		IF nSorterLogEnable.SORTER_DUMP THEN
			IF aSorterItems[nSorterClearIdx].ID <> '' THEN
				IF .nSorterLogEnable.SORTER_DUMP THEN
					sMessage := CONCAT(' Item: ', aSorterItems[nSorterClearIdx].ID);
					sMessage := CONCAT(sMessage,' Index: ');
					sMessage := CONCAT(sMessage, DINT_TO_STRING(nSorterClearIdx));
					// Write to the Error List
					ADSLOGSTR( msgCtrlMask := ADSLOG_MSGTYPE_HINT OR ADSLOG_MSGTYPE_LOG
						, msgFmtStr := 'Array Dump Info: %s'
						, strArg := sMessage);
				END_IF
			END_IF
		END_IF
		aSorterItems[nSorterClearIdx] := BlankItem;
	END_FOR
	ClearSorterArray := FALSE;
END_IF

// Setup and process the Sorter Encoder
st_SorterEncoder.EncoderRawCount := ENC_Raw;
st_SorterEncoder.BitMaskSize := SORTERMASKSIZE;
fb_SorterEncoder(Encoder := st_SorterEncoder, Simulate := bSimulate);

(*
	Initializes the Diverts.  
*)
{warning 'TODO: Fix references to Full and Confirm PE'}
{warning 'TODO: Add Configuration for all Diverts'}
aSorterDiverts[1].Config := aSorterDivertsCfgs[1];
aSorterDiverts[1].FullPE := TRUE;
aSorterDiverts[1].ConfirmPE := TRUE;

fb_CommissionSorterDiverts(
			//InductTrigger := Photoeyes.PE_22441.Out,
			ReferenceValue := st_SorterEncoder.CurrentCount, 
			//DischargeTrigger := Photoeyes.PE_23121.Out_OffFltrd,
			TestTime := T#10S, Diverts := aSorterDiverts);

// Provide a "hard-coded" default destination.
IF st_SorterCfg.DefaultDestination <= 0 THEN
	st_SorterCfg.DefaultDestination := 1;
END_IF						

// Name of the sorter equipment
//st_SorterCfg.Name := Conveyors.cfgP8005Label;
st_SorterCfg.DivertCount := NUMBEROFDIVERTS;
IF DivertToCommission > 0 THEN
	st_SorterCfg.DefaultDestination := DivertToCommission;
END_IF
st_Sorter.EncoderCounts := st_SorterEncoder.CurrentCount;
//st_Sorter.InductPE := PhotoEyes.PE_22441.Out_OnFltrd;
//st_Sorter.DischargePE := Photoeyes.PE_23081.Out_OnFltrd;

// Test the Encoder
//tEncoderOK.IN := (Conveyors.P8005_VFD.IsRunning AND (st_Sorter.EncoderCounts = nLastEncoderCount));
tEncoderOK(PT:=T#1S);

// OK when Q is not on, but the alarm is reversed
//GVL_IO.ENC_11321_OK := tEncoderOK.Q;

// Publish the sorter name
//GVL_IO.SorterName := st_SorterCfg.Name;

// Sorter
(*
	ProcessBuffers processes all associated buffers (Sorter/Divert/Arrival/Transport/Update)
	Items arriving at the sorter are detected and processed in this function block then deliverd to the SorterProgram
	Items inducted into sorter produce TransportResponse messages in this function block
	Items diverted off the sorter produce TransportComplete messages in this function block
*)
ProcessBuffers(st_NextToInduct := st_ToInduct
				, st_TempInductItem := st_TempItem
				, st_UpdateItem := st_Inducting
				, st_Sorter := st_Sorter
				, aDiverts := aSorterDiverts
				, aItems := aSorterItems
				, DivertToCommission := DivertToCommission
				, ItemsArrayMax := SORTERENCODERMAX
				, ItemsArrayMin := SORTERENCODERMIN);

// Capture rising and falling edge Triggers of the configured Sorter PE (Induct/Discharge)
rInductPE(CLK:= st_Sorter.InductPE, Q =>);
fInductPE(CLK:= st_Sorter.InductPE, Q =>);
rDischargePE(CLK:= st_Sorter.DischargePE, Q =>);
fDischargePE(CLK:= st_Sorter.DischargePE, Q =>);

// Prepare a dummy record for items that arrive before BCR data is received
// On the rising edge of the Induct PE
IF rInductPE.Q THEN
	IF .nSorterLogEnable.SORTER_INDUCT_PE THEN
		// Write to the Error List
		ADSLOGSTR( msgCtrlMask := ADSLOG_MSGTYPE_HINT OR ADSLOG_MSGTYPE_LOG
			, msgFmtStr := 'Induct PE Blocked : %s'
			, strArg := BOOL_TO_STRING(st_Sorter.InductPE)); 
	END_IF
	// Test for a UniqueID, which indicates that a Barcode has been received
	IF st_ToInduct.Item.UniqueID = 0 THEN
		// Capture and create relevant info
		st_TempItem.Counts := st_Sorter.EncoderCounts;
		st_TempItem.Item.UniqueID :=  UDINT_TO_DINT(st_Sorter.EncoderCounts);
		st_TempItem.Item.ID :=  CONCAT('T-', UDINT_TO_STRING(st_Sorter.EncoderCounts));
		st_TempItem.Item.Destination := st_SorterCfg.DefaultDestination;
		st_TempItem.Item.Status := E_StatusCode.UnidentifiedItem;
		IF .nSorterLogEnable.SORTER_TEMPID THEN
			ADSLOGSTR( msgCtrlMask := ADSLOG_MSGTYPE_HINT OR ADSLOG_MSGTYPE_LOG
				, msgFmtStr := 'Temp ID Assigned : %s'
				, strArg := st_TempItem.Item.ID);
		END_IF
	END_IF	
END_IF

// Clear the dummy record when the PE clears
// Items can only be inducted when the BCR info is received before or while the induct PE is blocked
IF fInductPE.Q THEN
	IF .nSorterLogEnable.SORTER_INDUCT_PE THEN
		// Write to the Error List
		ADSLOGSTR( msgCtrlMask := ADSLOG_MSGTYPE_HINT OR ADSLOG_MSGTYPE_LOG
			, msgFmtStr := 'Induct PE Blocked : %s'
			, strArg := BOOL_TO_STRING(st_Sorter.InductPE));
	END_IF
	// Clear the record
	st_TempItem.Counts := 0;
	st_TempItem.Item :=  BlankItem;
END_IF

(*
	SorterProgram is a separate Program
	Config portion of the st_sorter is separate to allow it be be persistent.
*)
st_sorter.Config := st_sorterCfg;
SorterProgram(st_Sorter := st_Sorter
		, In_ItemToInduct := st_ToInduct.Item
		, In_InductingItem := st_Inducting.Item
		, aItems := aSorterItems
		, aDiverts := aSorterDiverts
		, st_tempItem := st_TempItem
		, ItemsArrayMax := SORTERENCODERMAX
		, ItemsArrayMin := SORTERENCODERMIN
		, DivertArrayMax := DIVERTMIN
		, DivertArrayMin := NUMBEROFDIVERTS
		, st_DischargeItem => SorterDischargeItem);

// Log the diverts
FB_DivertLog(DivertArray := aSorterDiverts,
				DivertLogEnable := .nDivertLogEnable,
				EncoderCounts := st_SorterEncoder.CurrentCount);

END_PROGRAM

// ---- FunctionBlocks/Sorter/SorterProgram.TcPOU
PROGRAM SorterProgram

VAR_IN_OUT
	In_ItemToInduct					: ST_Item;
	In_InductingItem				: ST_Item;
	st_tempItem						: ST_ItemTemporary;	// Temporary record used when barcode not yet received
	st_Sorter						: ST_Sorter;
	aDiverts						: ARRAY[SorterExample.DIVERTMIN..SorterExample.NUMBEROFDIVERTS] OF ST_DIVERT;
	aItems 							: ARRAY[SorterExample.SORTERENCODERMIN..SorterExample.SORTERENCODERMAX] OF ST_Item;
END_VAR

VAR_INPUT
	ItemsArrayMax		: UDINT;
	ItemsArrayMin		: UDINT;
	DivertArrayMax		: DINT;
	DivertArrayMin		: DINT;
END_VAR

VAR_OUTPUT
	st_DischargeItem	:	ST_Item;
END_VAR
VAR
	// Sorter Diagnostics
	aSorterDiagLog		: ST_ItemLogBuffer;
	fbSorterDiagLog		: FB_ItemLogBuffer;

	//Logging Variables
	UpdateSorterLog : FB_UpdateLog;
	
	//Induct Variables
	testEncoderCount		: UDINT;
	exitEncoderCount		: UDINT;
	lastCompareCount		: UDINT;
	updatingEncoderCount	: UDINT;

	tailendcount		: DINT := 0;
	inductindex 		: DINT;
	
	//Divert Variables
	fb_DivertDecision 		: FB_DivertDecision;
	fb_DivertFullMonitor  	: FB_DivertFullMonitor;
	DivertIndex				: DINT;
	Divertoffset			: INT;
	nTestItemIndex			: UDINT;
	Output2ItemIndex		: UDINT;

